(* IEC 61131-3 sources: beebread/doc (part 9) *)

// Commented out for beedance: it uses TN_INPUT_MENU_POPUP, which is commented out.
// FUNCTION_BLOCK TN_INPUT_SELECT_POPUP
// VAR
// 	in_index : INT;
// 	in_Element_Count : INT;
// 	by_Cur_Key : BYTE;
// 	by_Attr : BYTE;
// 	st_String : STRING;
// END_VAR
// VAR
// 	us_TN_MENU_POPUP : us_TN_MENU_POPUP;
// 	FB_TN_INPUT_MENU_POPUP : TN_INPUT_MENU_POPUP;
// 	FB_TN_SC_WRITE : TN_SC_WRITE;
// END_VAR
// VAR_IN_OUT
// 	Xus_TN_SCREEN : us_TN_SCREEN;
// 	Xus_TN_INPUT_CONTROL_DATA : us_TN_INPUT_CONTROL_DATA;
// END_VAR
//
// (* evaluate user input -> selection text n *)
// IF (Xus_TN_INPUT_CONTROL_DATA.bo_Focus = TRUE) THEN
//
// 	by_Cur_Key := Xus_TN_INPUT_CONTROL_DATA.by_Input_Exten_Code;
//
// 	IF (us_TN_MENU_POPUP.bo_Activ = FALSE) THEN
// 		us_TN_MENU_POPUP.by_Input_Exten_Code := BYTE#00;
//
// 		(* evaluate return key *)
// 		IF (by_Cur_Key = BYTE#13) THEN
// 			(* pass popup menu parameters *)
// 			us_TN_MENU_POPUP.in_Y := Xus_TN_INPUT_CONTROL_DATA.in_Y;
// 			us_TN_MENU_POPUP.in_X := Xus_TN_INPUT_CONTROL_DATA.in_X;
// 			us_TN_MENU_POPUP.by_Attr_mF := Xus_TN_INPUT_CONTROL_DATA.by_Attr_mF;
// 			us_TN_MENU_POPUP.by_Attr_oF := Xus_TN_INPUT_CONTROL_DATA.by_Attr_oF;
// 			us_TN_MENU_POPUP.st_Menu_Text := Xus_TN_INPUT_CONTROL_DATA.st_Input_Data;
// 			us_TN_MENU_POPUP.bo_Create := TRUE;
// 			us_TN_MENU_POPUP.in_Cur_Item := INT#00;
// 		END_IF;
//
// 		IF (us_TN_MENU_POPUP.in_Cur_Item > INT#00) THEN
// 			Xus_TN_INPUT_CONTROL_DATA.in_selected := us_TN_MENU_POPUP.in_Cur_Item;
// 			Xus_TN_INPUT_CONTROL_DATA.bo_Input_Entered := TRUE;
// 			Xus_TN_INPUT_CONTROL_DATA.bo_Update_Input := TRUE;
// 			us_TN_MENU_POPUP.in_Cur_Item := INT#00;
// 		END_IF;
//
// 	ELSE
// 		us_TN_MENU_POPUP.by_Input_Exten_Code := by_Cur_Key;
// 	END_IF;
//
// 	(* call popup menu cyclically *)
// 	FB_TN_INPUT_MENU_POPUP(Xus_TN_MENU_POPUP := us_TN_MENU_POPUP, Xus_TN_SCREEN := Xus_TN_SCREEN);
//
// END_IF;
//
// (* update of the display *)
// IF (Xus_TN_INPUT_CONTROL_DATA.bo_Update_Input = TRUE) OR (Xus_TN_INPUT_CONTROL_DATA.bo_Update_All = TRUE) THEN
//
// 	(* output title text *)
// 	IF Xus_TN_INPUT_CONTROL_DATA.bo_Update_All = TRUE THEN
//
// 		IF (Xus_TN_INPUT_CONTROL_DATA.in_Title_X_Offset = INT#00) AND (Xus_TN_INPUT_CONTROL_DATA.in_Title_Y_Offset = INT#00) THEN
// 			(* if offset X,Y = 0 then position the title string left of the element *)
// 			FB_TN_SC_WRITE.Iin_Y := Xus_TN_INPUT_CONTROL_DATA.in_Y;
// 			FB_TN_SC_WRITE.Iin_X := Xus_TN_INPUT_CONTROL_DATA.in_X - LEN(Xus_TN_INPUT_CONTROL_DATA.st_Title_String);
//
// 		ELSE
// 			(* output title text via row, color offset *)
// 			FB_TN_SC_WRITE.Iin_Y := Xus_TN_INPUT_CONTROL_DATA.in_Y + Xus_TN_INPUT_CONTROL_DATA.in_Title_Y_Offset;
// 			FB_TN_SC_WRITE.Iin_X := Xus_TN_INPUT_CONTROL_DATA.in_X + Xus_TN_INPUT_CONTROL_DATA.in_Title_X_Offset;
// 		END_IF;
//
// 		(* output title text via row, color offset *)
// 		FB_TN_SC_WRITE(	Iby_ATTR := Xus_TN_INPUT_CONTROL_DATA.by_Title_Attr,
// 						Ist_STRING := Xus_TN_INPUT_CONTROL_DATA.st_Title_String,
// 						Xus_TN_SCREEN := Xus_TN_SCREEN);
// 	END_IF;
//
// 	in_Element_Count := ELEMENT_COUNT(SEP:=BYTE#35,ELEMENT:=Xus_TN_INPUT_CONTROL_DATA.st_Input_Data);
//
// 	IF in_Element_Count > INT#00 THEN
//
// 		Xus_TN_INPUT_CONTROL_DATA.in_selected:=LIMIT(1,Xus_TN_INPUT_CONTROL_DATA.in_selected,in_Element_Count);
//
// 		in_index := Xus_TN_INPUT_CONTROL_DATA.in_selected;
//
// 		st_String := ELEMENT_GET(SEP:=BYTE#35,POS:=in_index - 1,ELEMENT:=Xus_TN_INPUT_CONTROL_DATA.st_Input_Data);
//
// 		st_String:= FIX(str:=st_String,
// 						L:=LEN(Xus_TN_INPUT_CONTROL_DATA.st_Input_Mask),
// 						C:=BYTE#32,
// 						M:=Xus_TN_INPUT_CONTROL_DATA.in_Input_Option);
//
// 		Xus_TN_INPUT_CONTROL_DATA.st_Input_String := st_String;
//
// 		IF Xus_TN_INPUT_CONTROL_DATA.bo_Focus = TRUE THEN
// 			by_Attr := Xus_TN_INPUT_CONTROL_DATA.by_Attr_mF;
// 		ELSE
// 			by_Attr := Xus_TN_INPUT_CONTROL_DATA.by_Attr_oF;
// 		END_IF;
//
// 		FB_TN_SC_WRITE(	Iin_X := Xus_TN_INPUT_CONTROL_DATA.in_X,
// 								Iin_Y := Xus_TN_INPUT_CONTROL_DATA.in_Y,
// 								Iby_ATTR := by_Attr,
// 								Ist_STRING := st_String,
// 								Xus_TN_SCREEN := Xus_TN_SCREEN );
// 	END_IF;
//
// 	(* set cursor to current position *)
// 	Xus_TN_INPUT_CONTROL_DATA.in_Cursor_X := Xus_TN_INPUT_CONTROL_DATA.in_X;
// 	Xus_TN_INPUT_CONTROL_DATA.in_Cursor_Y := Xus_TN_INPUT_CONTROL_DATA.in_Y;
//
// 	(* reset update flags *)
// 	Xus_TN_INPUT_CONTROL_DATA.bo_Update_All   := FALSE;
// 	Xus_TN_INPUT_CONTROL_DATA.bo_Update_Input := FALSE;
//
// END_IF;
// END_FUNCTION_BLOCK

// Commented out for beedance: it uses ELEMENT_COUNT, which is commented out.
// FUNCTION_BLOCK TN_INPUT_SELECT_TEXT
// VAR
// 	in_count : INT;
// 	by_Attr : BYTE;
// 	st_String : STRING;
// END_VAR
// VAR
// 	FB_TN_SC_WRITE : TN_SC_WRITE;
// END_VAR
// VAR_IN_OUT
// 	Xus_TN_SCREEN : us_TN_SCREEN;
// 	Xus_TN_INPUT_CONTROL_DATA : us_TN_INPUT_CONTROL_DATA;
// END_VAR
//
// (* evaluate user input -> selection text n *)
// IF Xus_TN_INPUT_CONTROL_DATA.bo_Focus = TRUE THEN
//
// (* evaluate space key *)
// 	IF Xus_TN_INPUT_CONTROL_DATA.by_Input_ASCII_Code = BYTE#32 THEN
// 		Xus_TN_INPUT_CONTROL_DATA.in_selected := Xus_TN_INPUT_CONTROL_DATA.in_selected + INT#01;
// 		Xus_TN_INPUT_CONTROL_DATA.bo_Update_Input := TRUE;
// 	END_IF;
//
// 	(* evaluate return key *)
// 	IF Xus_TN_INPUT_CONTROL_DATA.by_Input_Exten_Code = BYTE#13 THEN
// 		Xus_TN_INPUT_CONTROL_DATA.bo_Input_Entered := TRUE;
// 	END_IF;
//
// END_IF;
//
// (* update of the display *)
// IF (Xus_TN_INPUT_CONTROL_DATA.bo_Update_Input = TRUE) OR (Xus_TN_INPUT_CONTROL_DATA.bo_Update_All = TRUE) THEN
//
// 	(* output title text *)
// 	IF Xus_TN_INPUT_CONTROL_DATA.bo_Update_All = TRUE THEN
//
// 		IF (Xus_TN_INPUT_CONTROL_DATA.in_Title_X_Offset = INT#00) AND (Xus_TN_INPUT_CONTROL_DATA.in_Title_Y_Offset = INT#00) THEN
// 			(* if offset X,Y = 0 then position the title string left of the element *)
// 			FB_TN_SC_WRITE.Iin_Y := Xus_TN_INPUT_CONTROL_DATA.in_Y;
// 			FB_TN_SC_WRITE.Iin_X := Xus_TN_INPUT_CONTROL_DATA.in_X - LEN(Xus_TN_INPUT_CONTROL_DATA.st_Title_String);
//
// 		ELSE
// 			(* output title text via row, color offset *)
// 			FB_TN_SC_WRITE.Iin_Y := Xus_TN_INPUT_CONTROL_DATA.in_Y + Xus_TN_INPUT_CONTROL_DATA.in_Title_Y_Offset;
// 			FB_TN_SC_WRITE.Iin_X := Xus_TN_INPUT_CONTROL_DATA.in_X + Xus_TN_INPUT_CONTROL_DATA.in_Title_X_Offset;
// 		END_IF;
//
// 		(* output title text via row, color offset *)
// 		FB_TN_SC_WRITE(	Iby_ATTR := Xus_TN_INPUT_CONTROL_DATA.by_Title_Attr,
// 						Ist_STRING := Xus_TN_INPUT_CONTROL_DATA.st_Title_String,
// 						Xus_TN_SCREEN := Xus_TN_SCREEN);
//
// 	END_IF;
//
// 	(* process input line *)
//
// 	(* determine number of elements *)
// 	in_count := ELEMENT_COUNT(SEP:=BYTE#35,ELEMENT:=Xus_TN_INPUT_CONTROL_DATA.st_Input_Data);
//
// 	IF in_Count > INT#00 THEN
//
// 		IF Xus_TN_INPUT_CONTROL_DATA.in_selected < INT#1 THEN
// 			Xus_TN_INPUT_CONTROL_DATA.in_selected := INT#01;
// 		END_IF;
//
// 		IF Xus_TN_INPUT_CONTROL_DATA.in_selected > in_count THEN
// 			Xus_TN_INPUT_CONTROL_DATA.in_selected := INT#01;
// 		END_IF;
//
// 		st_String := ELEMENT_GET(SEP:=BYTE#35,POS:=Xus_TN_INPUT_CONTROL_DATA.in_selected - 1,ELEMENT:=Xus_TN_INPUT_CONTROL_DATA.st_Input_Data);
//
// 		st_String := FIX(	str:=st_String,
// 							L:=LEN(Xus_TN_INPUT_CONTROL_DATA.st_Input_Mask),
// 							C:=BYTE#32,
// 							M:=Xus_TN_INPUT_CONTROL_DATA.in_Input_Option);
//
// 		Xus_TN_INPUT_CONTROL_DATA.st_Input_String := st_String;
//
// 		IF Xus_TN_INPUT_CONTROL_DATA.bo_Focus = TRUE THEN
// 			by_Attr := Xus_TN_INPUT_CONTROL_DATA.by_Attr_mF;
// 		ELSE
// 			by_Attr := Xus_TN_INPUT_CONTROL_DATA.by_Attr_oF;
// 		END_IF;
//
// 		FB_TN_SC_WRITE(	Iin_Y := Xus_TN_INPUT_CONTROL_DATA.in_Y,
// 						Iin_X := Xus_TN_INPUT_CONTROL_DATA.in_X,
// 						Iby_ATTR := by_Attr,
// 						Ist_STRING := st_String,
// 						Xus_TN_SCREEN := Xus_TN_SCREEN);
// 	END_IF;
//
// 	(* set cursor to current position *)
// 	Xus_TN_INPUT_CONTROL_DATA.in_Cursor_Y := Xus_TN_INPUT_CONTROL_DATA.in_Y;
// 	Xus_TN_INPUT_CONTROL_DATA.in_Cursor_X := Xus_TN_INPUT_CONTROL_DATA.in_X;
//
// 	(* reset update flags *)
// 	Xus_TN_INPUT_CONTROL_DATA.bo_Update_All := FALSE;
// 	Xus_TN_INPUT_CONTROL_DATA.bo_Update_Input := FALSE;
//
// END_IF;
// END_FUNCTION_BLOCK

FUNCTION_BLOCK TN_RECEIVE
VAR_IN_OUT
	R_BUF :	NETWORK_BUFFER;
	Xus_TN_SCREEN : us_TN_SCREEN;
END_VAR
VAR
	REQ_Size : UINT;
	REQ1 : BYTE;
	REQ2 : BYTE;
	REQ3 : BYTE;
END_VAR

(* evaluate data reception *)
Xus_TN_SCREEN.by_Input_ASCII_Code := BYTE#00;
Xus_TN_SCREEN.by_Input_Exten_Code := BYTE#00;

IF R_BUF.SIZE > UINT#0 THEN
	(* evaluate received data *)
	REQ_Size := R_BUF.SIZE;
	REQ1 := R_BUF.BUFFER[0];
	REQ2 := R_BUF.BUFFER[1];
	REQ3 := R_BUF.BUFFER[2];

	IF REQ1 = BYTE#27 AND REQ_Size >= UINT#3 THEN (* Escape *)
		IF REQ2 = BYTE#91 THEN (* Cursor code *)
			IF (REQ3 >= BYTE#65 AND REQ3 <= BYTE#68) OR (REQ3 = BYTE#72) OR (REQ3 = BYTE#75) THEN (* 65..68 = cursor up,down,right,left / 72 = HOME / 75 = END *)
				Xus_TN_SCREEN.by_Input_Exten_Code := REQ3;
			END_IF;
		ELSIF REQ2 = BYTE#79 THEN (* special keys F1/F2/F3/F4 *)
			IF REQ3 >= BYTE#80 AND REQ3 <= BYTE#83 THEN
				Xus_TN_SCREEN.by_Input_Exten_Code := REQ3;
			END_IF;
		END_IF;
	ELSIF REQ1 >= BYTE#32 AND REQ1 <= BYTE#126 THEN
		Xus_TN_SCREEN.by_Input_ASCII_Code := REQ1;
		Xus_TN_SCREEN.bo_Input_ASCII_IsNum := ISC_NUM(REQ1); (* check for numeric input *)
	ELSIF REQ1 = BYTE#8 OR REQ1 = BYTE#9 OR REQ1 = BYTE#13 OR REQ1 = BYTE#27 THEN (* check for control characters 8=Backspace / 9=Tab / 13=Return / 27=Escape *)
		Xus_TN_SCREEN.by_Input_Exten_Code := REQ1;
	END_IF;

	(* set receive buffer data length to zero (destroy telegram *)
	R_BUF.SIZE := UINT#00;
END_IF;
END_FUNCTION_BLOCK

FUNCTION_BLOCK TN_SC_ADD_SHADOW
VAR
	in_Offset : INT;
	in_X : INT;
	in_Y : INT;
END_VAR
VAR_INPUT
	Iin_Y1 : INT;
	Iin_X1 : INT;
	Iin_Y2 : INT;
	Iin_X2 : INT;
	Iin_OPTION : INT;
END_VAR
VAR_IN_OUT
	Xus_TN_SCREEN : us_TN_SCREEN;
END_VAR

IF TN_SC_XY2_ERROR(Iin_X1,Iin_Y1,Iin_X2,Iin_Y2) THEN RETURN; END_IF;

IF Iin_Y1 < 0 OR Iin_X1 < 0 OR Iin_Y2 < 0 OR Iin_X2 < 0 THEN RETURN; END_IF; (* check min values *)
IF Iin_Y1 > 23 OR Iin_X1 > 79 OR Iin_Y2 > 23 OR Iin_X2 > 79 THEN RETURN; END_IF; (* check max values *)

in_Offset := (Iin_Y1 * 80) + Iin_X2;

IF Iin_OPTION = INT#00 THEN
	(* create shadow by adjusting color *)
	FOR in_Y := Iin_Y1 TO Iin_Y2 DO
		Xus_TN_SCREEN.bya_COLOR[in_Offset] := TN_SC_SHADOW_ATTR(Xus_TN_SCREEN.bya_COLOR[in_Offset]);
		in_Offset := in_Offset + 80;
		Xus_TN_SCREEN.bya_Line_Update[in_Y] := TRUE; (* mark line for update *)
	END_FOR;
ELSE
	(* create shadow with black color and spaces *)
	FOR in_Y := Iin_Y1 TO Iin_Y2 DO
		Xus_TN_SCREEN.bya_COLOR[in_Offset] := BYTE#00;
		Xus_TN_SCREEN.bya_CHAR[in_Offset] := BYTE#32;
		in_Offset := in_Offset + 80;
		Xus_TN_SCREEN.bya_Line_Update[in_Y] := TRUE; (* mark line for update *)
	END_FOR;
END_IF;

in_Offset := (Iin_Y2 * 80) + Iin_X1;

IF Iin_OPTION = INT#00 THEN
	(* create shadow by adjusting color *)
	FOR in_X  := Iin_X1 TO Iin_X2 DO
		Xus_TN_SCREEN.bya_COLOR[in_Offset] := TN_SC_SHADOW_ATTR(Xus_TN_SCREEN.bya_COLOR[in_Offset]);
		in_Offset := in_Offset + 1;
	END_FOR;
ELSE
	(* create shadow with black color and spaces *)
	FOR in_X  := Iin_X1 TO Iin_X2 DO
		Xus_TN_SCREEN.bya_COLOR[in_Offset] := BYTE#00;
		Xus_TN_SCREEN.bya_CHAR[in_Offset] := BYTE#32;
		in_Offset := in_Offset + 1;
	END_FOR;
END_IF;
END_FUNCTION_BLOCK

FUNCTION_BLOCK TN_SC_AREA_RESTORE
VAR
	in_Offset_1 : INT;
	in_Offset_2 : INT;
	in_Y : INT;
	in_X : INT;
	in_Y1 : INT;
	in_X1 : INT;
	in_Y2 : INT;
	in_X2 : INT;
END_VAR
VAR_IN_OUT
	Xus_TN_SCREEN : us_TN_SCREEN;
END_VAR

IF Xus_TN_SCREEN.bya_BACKUP[0] > BYTE#00 THEN

	(* read parameters *)
	in_X1 := BYTE_TO_INT(Xus_TN_SCREEN.bya_BACKUP[1]);
	in_Y1 := BYTE_TO_INT(Xus_TN_SCREEN.bya_BACKUP[2]);
	in_X2 := BYTE_TO_INT(Xus_TN_SCREEN.bya_BACKUP[3]);
	in_Y2 := BYTE_TO_INT(Xus_TN_SCREEN.bya_BACKUP[4]);

	IF TN_SC_XY2_ERROR(in_X1,in_Y1,in_X2,in_Y2) THEN RETURN; END_IF;
	in_Offset_2 := 5;

	(* restore CHAR and COLOR from BUFFER *)
	FOR in_Y := in_Y1 TO in_Y2 DO

		Xus_TN_SCREEN.bya_Line_Update[in_Y] := TRUE; (* release line for update *)
		in_Offset_1 := (in_Y * 80) + in_X1;

		FOR in_X := in_X1 TO in_X2 DO

			Xus_TN_SCREEN.bya_CHAR[in_Offset_1] := Xus_TN_SCREEN.bya_BACKUP[in_Offset_2];
			in_Offset_2 := in_Offset_2 + INT#01;

			Xus_TN_SCREEN.bya_COLOR[in_Offset_1] := Xus_TN_SCREEN.bya_BACKUP[in_Offset_2];
			in_Offset_2 := in_Offset_2 + INT#01;
			in_Offset_1 := in_Offset_1 + INT#01;

		END_FOR;
	END_FOR;

	(* mark data as invalid *)
	Xus_TN_SCREEN.bya_BACKUP[0] := BYTE#00;
END_IF;
END_FUNCTION_BLOCK

FUNCTION_BLOCK TN_SC_AREA_SAVE
VAR
	in_Offset_1 : INT;
	in_Offset_2 : INT;
	in_Y : INT;
	in_X : INT;
END_VAR
VAR_INPUT
	Iin_Y1 : INT;
	Iin_X1 : INT;
	Iin_Y2 : INT;
	Iin_X2 : INT;
END_VAR
VAR_IN_OUT
	Xus_TN_SCREEN : us_TN_SCREEN;
END_VAR

IF TN_SC_XY2_ERROR(Iin_X1,Iin_Y1,Iin_X2,Iin_Y2) THEN RETURN; END_IF;

(* store parameters *)
Xus_TN_SCREEN.bya_BACKUP[0] := BYTE#1;
Xus_TN_SCREEN.bya_BACKUP[1] := INT_TO_BYTE(Iin_X1);
Xus_TN_SCREEN.bya_BACKUP[2] := INT_TO_BYTE(Iin_Y1);
Xus_TN_SCREEN.bya_BACKUP[3] := INT_TO_BYTE(Iin_X2);
Xus_TN_SCREEN.bya_BACKUP[4] := INT_TO_BYTE(Iin_Y2);

in_Offset_2 := 5;
(* save CHAR and COLOR in BUFFER *)
FOR in_Y := Iin_Y1 TO Iin_Y2 DO

	in_Offset_1 := (in_Y * 80) + Iin_X1;
	FOR in_X := Iin_X1 TO Iin_X2 DO
		Xus_TN_SCREEN.bya_BACKUP[in_Offset_2] := Xus_TN_SCREEN.bya_CHAR[in_Offset_1];
		in_Offset_2 := in_Offset_2 + INT#01;
		Xus_TN_SCREEN.bya_BACKUP[in_Offset_2] := Xus_TN_SCREEN.bya_COLOR[in_Offset_1];
		in_Offset_2 := in_Offset_2 + INT#01;
		in_Offset_1 := in_Offset_1 + INT#01;
	END_FOR;
END_FOR;
END_FUNCTION_BLOCK

FUNCTION_BLOCK TN_SC_BOX
VAR
	FB_TN_SC_FILL : TN_SC_FILL;
	by_BorderChar_L_T : BYTE;
	by_BorderChar_T : BYTE;
	by_BorderChar_B : BYTE;
	by_BorderChar_R_T : BYTE;
	by_BorderChar_L : BYTE;
	by_BorderChar_R : BYTE;
	by_BorderChar_L_B : BYTE;
	by_BorderChar_R_B : BYTE;
	in_Y : INT;
	in_X : INT;
	in_Border_Offset : INT;
	in_Offset_1 : INT;
	in_Offset_2 : INT;
END_VAR
VAR_INPUT
	Iin_Y1 : INT;
	Iin_X1 : INT;
	Iin_Y2 : INT;
	Iin_X2 : INT;
	Iby_FILL : BYTE;
	Iby_ATTR : BYTE;
	Iin_BORDER : INT;
END_VAR
VAR_IN_OUT
	Xus_TN_SCREEN : us_TN_SCREEN;
END_VAR

IF TN_SC_XY2_ERROR(Iin_X1,Iin_Y1,Iin_X2,Iin_Y2) THEN RETURN; END_IF;

(* determine border type *)
CASE Iin_Border OF
0:
	in_Border_Offset := 0;
1:
	by_BorderChar_L_T := BYTE#218; (* top left *)
	by_BorderChar_T := BYTE#196; (* top *)
	by_BorderChar_R_T := BYTE#191; (* top right *)
	by_BorderChar_L := BYTE#179; (* left *)
	by_BorderChar_R := BYTE#179; (* right *)
	by_BorderChar_B := BYTE#196; (* bottom *)
	by_BorderChar_L_B := BYTE#217; (* bottom left *)
	by_BorderChar_R_B := BYTE#192; (* bottom right *)
	in_Border_Offset := 1;
 2:
	by_BorderChar_L_T := BYTE#201;
	by_BorderChar_T := BYTE#205;
	by_BorderChar_R_T := BYTE#187;
	by_BorderChar_L := BYTE#186;
	by_BorderChar_R := BYTE#186;
	by_BorderChar_B := BYTE#205;
	by_BorderChar_L_B := BYTE#188;
	by_BorderChar_R_B := BYTE#200;
	in_Border_Offset := 1;
ELSE
	by_BorderChar_L_T := BYTE#32;
	by_BorderChar_T := BYTE#32;
	by_BorderChar_R_T := BYTE#32;
	by_BorderChar_L := BYTE#32;
	by_BorderChar_R := BYTE#32;
	by_BorderChar_B := BYTE#32;
	by_BorderChar_L_B := BYTE#32;
	by_BorderChar_R_B := BYTE#32;
	in_Border_Offset := 1;

END_CASE;

IF Iby_FILL > BYTE#0 THEN (* FILL character present? -> draw box *)

	(* draw fill function one character row smaller *)
	FB_TN_SC_FILL(	Iin_Y1 := Iin_Y1 + in_Border_Offset,
					Iin_X1 := Iin_X1 + in_Border_Offset,
					Iin_Y2 := Iin_Y2 - in_Border_Offset,
					Iin_X2 := Iin_X2 - in_Border_Offset,
					Iby_CHAR := Iby_FILL,
					Iby_Attr := Iby_ATTR,
					Xus_TN_SCREEN := Xus_TN_SCREEN);
END_IF;

IF Iin_BORDER = 0 THEN RETURN; END_IF;

(* output left and right border *)

in_Offset_1 := (Iin_Y1 * 80) + Iin_X1;
in_Offset_2 := (Iin_Y1 * 80) + Iin_X2;

FOR in_Y := Iin_Y1 TO Iin_Y2 DO

	(* release line for update *)
	Xus_TN_SCREEN.bya_Line_Update[in_Y] := TRUE;

	Xus_TN_SCREEN.bya_CHAR[in_Offset_1] := by_BorderChar_L;
	Xus_TN_SCREEN.bya_COLOR[in_Offset_1] := Iby_Attr;

	Xus_TN_SCREEN.bya_CHAR[in_Offset_2] := by_BorderChar_R;
	Xus_TN_SCREEN.bya_COLOR[in_Offset_2] := Iby_Attr;

	in_Offset_1 := in_Offset_1 + 80;
	in_Offset_2 := in_Offset_2 + 80;

END_FOR;

(* output bottom and top border *)
in_Offset_1 := (Iin_Y1 * 80) + Iin_X1;
in_Offset_2 := (Iin_Y2 * 80) + Iin_X1;

FOR in_X := Iin_X1 TO Iin_X2 DO

	Xus_TN_SCREEN.bya_CHAR[in_Offset_1] := by_BorderChar_T;
	Xus_TN_SCREEN.bya_COLOR[in_Offset_1] := Iby_Attr;

	Xus_TN_SCREEN.bya_CHAR[in_Offset_2] := by_BorderChar_B;
	Xus_TN_SCREEN.bya_COLOR[in_Offset_2] := Iby_Attr;

	in_Offset_1 := in_Offset_1 + INT#1;
	in_Offset_2 := in_Offset_2 + INT#1;

END_FOR;

(* output top left corner *)
in_Offset_1 := (Iin_Y1 * 80) + Iin_X1;
Xus_TN_SCREEN.bya_CHAR[in_Offset_1] := by_BorderChar_L_T;
Xus_TN_SCREEN.bya_COLOR[in_Offset_1] := Iby_Attr;

(* output top right corner *)
in_Offset_1 := (Iin_Y1 * 80) + Iin_X2;
Xus_TN_SCREEN.bya_CHAR[in_Offset_1] := by_BorderChar_R_T;
Xus_TN_SCREEN.bya_COLOR[in_Offset_1] := Iby_Attr;

(* output bottom left corner *)
in_Offset_1 := (Iin_Y2 * 80) + Iin_X1;
Xus_TN_SCREEN.bya_CHAR[in_Offset_1] := by_BorderChar_R_B;
Xus_TN_SCREEN.bya_COLOR[in_Offset_1] := Iby_Attr;

(* output bottom right corner *)
in_Offset_1 := (Iin_Y2 * 80) + Iin_X2;
Xus_TN_SCREEN.bya_CHAR[in_Offset_1] := by_BorderChar_L_B;
Xus_TN_SCREEN.bya_COLOR[in_Offset_1] := Iby_Attr;
END_FUNCTION_BLOCK

FUNCTION_BLOCK TN_SC_FILL
VAR
	in_X : INT;
	in_Y : INT;
	in_Offset : INT;
END_VAR
VAR_INPUT
	Iin_Y1 : INT;
	Iin_X1 : INT;
	Iin_Y2 : INT;
	Iin_X2 : INT;
	Iby_CHAR : BYTE;
	Iby_Attr : BYTE;
END_VAR
VAR_IN_OUT
	Xus_TN_SCREEN : us_TN_SCREEN;
END_VAR

IF TN_SC_XY2_ERROR(Iin_X1,Iin_Y1,Iin_X2,Iin_Y2) THEN RETURN; END_IF;

FOR in_Y := Iin_Y1 TO Iin_Y2 DO
	Xus_TN_SCREEN.bya_Line_Update[in_Y] := TRUE; (* release line for update *)
	in_Offset := (in_Y * 80) + Iin_X1;
	FOR in_X := Iin_X1 TO Iin_X2 DO
		Xus_TN_SCREEN.bya_CHAR[in_Offset]  := Iby_CHAR; (* enter character *)
		Xus_TN_SCREEN.bya_COLOR[in_Offset] := Iby_Attr; (* enter color *)
		in_Offset := in_Offset + 1;
	END_FOR;
END_FOR;
END_FUNCTION_BLOCK

FUNCTION_BLOCK TN_SC_LINE
VAR
	by_Connect_Left_Char : BYTE;
	by_Connect_Right_Char : BYTE;
	by_Connect_Top_Char : BYTE;
	by_Connect_Bottom_Char : BYTE;
	by_Connect_Cruz_Char : BYTE;
	by_Vertikal_Line_Char : BYTE;
	by_Horzontal_Line_Char : BYTE;
	by_old_Char : BYTE;
	in_Offset_1 : INT;
	in_ROW_Index : INT;
	in_COL_Index : INT;
	by_Char : BYTE;
END_VAR
VAR_INPUT
	Iin_X1 : INT;
	Iin_Y1 : INT;
	Iin_X2 : INT;
	Iin_Y2 : INT;
	Iby_ATTR : BYTE;
	Iby_BORDER : BYTE;
END_VAR
VAR_IN_OUT
	Xus_TN_SCREEN : us_TN_SCREEN;
END_VAR

IF TN_SC_XY2_ERROR(Iin_X1,Iin_Y1,Iin_X2,Iin_Y2) THEN RETURN; END_IF;

(* determine border type *)
IF Iby_Border = BYTE#01 THEN (* Single Line *)
	by_Connect_Top_Char := BYTE#16#C2;
	by_Connect_Bottom_Char := BYTE#16#C1;
	by_Connect_Left_Char := BYTE#16#C3;
	by_Connect_Right_Char := BYTE#16#B4;
	by_Horzontal_Line_Char := BYTE#16#C4;
	by_Vertikal_Line_Char := BYTE#16#B3;
	by_Connect_Cruz_Char := BYTE#16#C5;
ELSIF Iby_Border = BYTE#02 THEN	(* double line *)
	by_Connect_Top_Char := BYTE#16#CB;
	by_Connect_Bottom_Char := BYTE#16#CA;
	by_Connect_Left_Char := BYTE#16#CC;
	by_Connect_Right_Char := BYTE#16#B9;
	by_Horzontal_Line_Char := BYTE#16#CD;
	by_Vertikal_Line_Char := BYTE#16#BA;
	by_Connect_Cruz_Char := BYTE#16#CE;
ELSE (* full line *)
	by_Connect_Top_Char := Iby_Border;
	by_Connect_Bottom_Char := Iby_Border;
	by_Connect_Left_Char := Iby_Border;
	by_Connect_Right_Char := Iby_Border;
	by_Horzontal_Line_Char := Iby_Border;
	by_Vertikal_Line_Char := Iby_Border;
	by_Connect_Cruz_Char := Iby_Border;
END_IF;

(* draw vertical line *)
IF Iin_X1 = Iin_X2 THEN
	in_Offset_1 := (Iin_Y1 * 80) + Iin_X1;
	FOR in_ROW_Index := Iin_Y1 TO Iin_Y2 DO
		by_old_Char := Xus_TN_SCREEN.bya_CHAR[in_Offset_1]; (* read existing character *)
		by_Char := by_Vertikal_Line_Char; (* preset default characters *)
		IF by_old_Char = by_Horzontal_Line_Char THEN (* intersection detected *)
			IF in_ROW_Index = Iin_Y1 THEN (* handle start of line *)
				by_Char := by_Connect_Top_Char;
			ELSIF in_ROW_Index = Iin_Y2 THEN (* handle end of line *)
				by_Char := by_Connect_Bottom_Char;
			ELSE (* handle crossing point *)
				by_Char := by_Connect_Cruz_Char;
			END_IF;
		END_IF;
		Xus_TN_SCREEN.bya_Line_Update[in_ROW_Index] := TRUE; (* release line for update *)
		Xus_TN_SCREEN.bya_CHAR[in_Offset_1] := by_Char;
		Xus_TN_SCREEN.bya_COLOR[in_Offset_1] := Iby_Attr;
		in_Offset_1 := in_Offset_1 + 80;
	END_FOR;

ELSIF Iin_Y1 = Iin_Y2 THEN (* draw horizontal line *)
	Xus_TN_SCREEN.bya_Line_Update[Iin_Y1] := TRUE; (* release line for update *)
	in_Offset_1 := (Iin_Y1 * 80) + Iin_X1;
	FOR in_COL_Index := Iin_X1 TO Iin_X2 DO
		by_old_Char := Xus_TN_SCREEN.bya_CHAR[in_Offset_1]; (* read existing character *)
		by_Char := by_Horzontal_Line_Char; (* preset default characters *)
		IF by_old_Char = by_Vertikal_Line_Char THEN (* intersection detected *)
			IF in_COL_Index = Iin_X1 THEN (* handle start of line *)
				by_Char := by_Connect_Left_Char;
			ELSIF in_COL_Index = Iin_X2 THEN (* handle end of line *)
				by_Char := by_Connect_Right_Char;
			ELSE (* handle crossing point *)
				by_Char := by_Connect_Cruz_Char;
			END_IF;
		END_IF;
		Xus_TN_SCREEN.bya_CHAR[in_Offset_1] := by_Char;
		Xus_TN_SCREEN.bya_COLOR[in_Offset_1] := Iby_Attr;
		in_Offset_1 := in_Offset_1 + 1;
	END_FOR;
END_IF;
END_FUNCTION_BLOCK

FUNCTION_BLOCK TN_SC_READ_ATTR
VAR
	in_Offset : INT;
END_VAR
VAR_INPUT
	Iin_Y : INT;
	Iin_X : INT;
END_VAR
VAR_OUTPUT
	Oby_ATTR : BYTE;
END_VAR
VAR_IN_OUT
	Xus_TN_SCREEN : us_TN_SCREEN;
END_VAR

IF TN_SC_XY_ERROR(Iin_X,Iin_Y) THEN RETURN; END_IF;
in_Offset := (Iin_Y * 80) + Iin_X;
Oby_ATTR := Xus_TN_SCREEN.bya_COLOR[in_Offset]; (* read attributes *)
END_FUNCTION_BLOCK

FUNCTION_BLOCK TN_SC_READ_CHAR
VAR
	in_Offset : INT;
END_VAR
VAR_INPUT
	Iin_Y : INT;
	Iin_X : INT;
END_VAR
VAR_OUTPUT
	Oby_CHAR : BYTE;
END_VAR
VAR_IN_OUT
	Xus_TN_SCREEN : us_TN_SCREEN;
END_VAR

IF TN_SC_XY_ERROR(Iin_X,Iin_Y) THEN RETURN; END_IF;
in_Offset := (Iin_Y * 80) + Iin_X;
Oby_CHAR := Xus_TN_SCREEN.bya_CHAR[in_Offset]; (* read character *)
END_FUNCTION_BLOCK

FUNCTION TN_SC_SHADOW_ATTR : BYTE
VAR_INPUT
	Iby_ATTR : BYTE;
END_VAR

(* change background color to black      *)
(* and switch on dark foreground colors *)
TN_SC_SHADOW_ATTR := ((Iby_ATTR AND BYTE#2#11110000) OR BYTE#2#00001000);
END_FUNCTION

// Commented out for beedance: it uses FIX, which is commented out.
// FUNCTION_BLOCK TN_SC_VIEWPORT
// VAR
// 	FB_TN_SC_WRITE : TN_SC_WRITE;
// 	FB_TON : TON;
// END_VAR
// VAR
// 	in_index : INT;
// 	in_Color : INT;
// 	by_Attr : BYTE;
// 	in_count : INT;
// END_VAR
// VAR_IN_OUT
// 	Xus_LOG_VIEWPORT : us_LOG_VIEWPORT;
// 	Xus_LOG_CONTROL : LOG_CONTROL;
// 	Xus_TN_SCREEN : us_TN_SCREEN;
// END_VAR
// VAR_INPUT
// 	Iin_X : INT;
// 	Iin_Y : INT;
// 	Iin_Width : INT;
// 	Idw_ATTR_1 : DWORD;
// 	Idw_ATTR_2 : DWORD;
// 	Iti_TIME : TIME;
// END_VAR
//
// (* output LOG messages *)
//
// IF Xus_LOG_VIEWPORT.UPDATE AND FB_TON.Q THEN (* update requested and delay time elapsed *)
// 	Xus_LOG_VIEWPORT.UPDATE := FALSE;
// 	FOR in_count := 1 TO Xus_LOG_VIEWPORT.COUNT DO (* process all viewport lines *)
// 		in_index := Xus_LOG_VIEWPORT.LINE_ARRAY[in_count];
// 		(* read color from the option parameter >0,Level,Back,Front< *)
// 		in_Color := DWORD_TO_INT(Xus_LOG_CONTROL.MSG_OPTION[in_index] AND DWORD#2#1111);
//
// 		CASE in_Color OF
// 		0..3: by_Attr := BYTE_OF_DWORD(Idw_ATTR_1,INT_TO_BYTE(in_Color));
// 		4..7: by_Attr := BYTE_OF_DWORD(Idw_ATTR_2,INT_TO_BYTE(in_Color));
// 		ELSE
// 			by_Attr := BYTE_OF_DWORD(Idw_ATTR_1,BYTE#0);
// 		END_CASE;
//
// 		(* output message (text + color) *)
// 		FB_TN_SC_WRITE(	Iin_Y := Iin_Y + in_count - INT#01,
// 						Iin_X := Iin_X,
// 						Iby_ATTR := by_Attr,
// 						Ist_STRING := FIX(str := Xus_LOG_CONTROL.MSG[in_index], L := Iin_Width, C := BYTE#32, M := INT#00), (* pad or truncate string on the right *)
// 						Xus_TN_SCREEN := Xus_TN_SCREEN);
//
// 	END_FOR;
//
// 	(* stop/reset timer *)
// 	FB_TON.IN := FALSE;
// 	FB_TON.PT := Iti_TIME;
// 	FB_TON();
//
// END_IF;
//
// (* update time delay *)
// FB_TON.IN := TRUE;
// FB_TON.PT := Iti_TIME;
// FB_TON();
// END_FUNCTION_BLOCK

// Commented out for beedance: it uses CODE, which is commented out.
// FUNCTION_BLOCK TN_SC_WRITE
// VAR
// 	bo_Color : BOOL;
// 	in_Offset : INT;
// 	in_Char_Index : INT;
// 	in_String_Length : INT;
// END_VAR
// VAR_INPUT
// 	Iin_Y : INT;
// 	Iin_X : INT;
// 	Iby_ATTR : BYTE;
// 	Ist_STRING : STRING;
// END_VAR
// VAR_IN_OUT
// 	Xus_TN_SCREEN : us_TN_SCREEN;
// END_VAR
//
// in_String_Length := LEN(Ist_STRING);
// IF TN_SC_XY_ERROR(Iin_X + in_String_Length - 1,Iin_Y) THEN RETURN; END_IF;
// Xus_TN_SCREEN.bya_Line_Update[Iin_Y] := TRUE; (* release line for update *)
// in_Offset := (Iin_Y * 80) + Iin_X; (* calculate offset of the first character *)
// bo_Color := Iby_ATTR <> BYTE#00;
//
// (* copy characters and attributes of the string *)
// FOR in_Char_Index := 1 TO in_String_Length DO
// 	IF bo_Color THEN Xus_TN_SCREEN.bya_COLOR[in_Offset] := Iby_ATTR; END_IF;
// 	Xus_TN_SCREEN.bya_CHAR[in_Offset] := CODE(STR:=Ist_STRING,POS:=in_Char_Index);
// 	in_Offset := in_Offset + INT#1;
// END_FOR;
//
// Xus_TN_SCREEN.in_EOS_Offset := in_Offset; (* save end of string offset *)
// END_FUNCTION_BLOCK

FUNCTION_BLOCK TN_SC_WRITE_ATTR
VAR
	in_Offset : INT;
END_VAR
VAR_INPUT
	Iin_Y : INT;
	Iin_X : INT;
	Iby_ATTR : BYTE;
END_VAR
VAR_IN_OUT
	Xus_TN_SCREEN : us_TN_SCREEN;
END_VAR

IF TN_SC_XY_ERROR(Iin_X,Iin_Y) THEN RETURN; END_IF;
in_Offset := (Iin_Y * 80) + Iin_X;
Xus_TN_SCREEN.bya_COLOR[in_Offset] := Iby_ATTR; (* write attributes *)
END_FUNCTION_BLOCK

// Commented out for beedance: it uses TN_SC_WRITE, which is commented out.
// FUNCTION_BLOCK TN_SC_WRITE_C
// VAR
// 	FB_TN_SC_WRITE : TN_SC_WRITE;
// END_VAR
// VAR_INPUT
// 	Iin_Y : INT;
// 	Iin_X : INT;
// 	Iby_ATTR : BYTE;
// 	Ist_STRING : STRING;
// 	Iin_LENGTH : INT;
// 	Iin_OPTION : INT;
// END_VAR
// VAR_IN_OUT
// 	Xus_TN_SCREEN : us_TN_SCREEN;
// END_VAR
//
// (* output text *)
// FB_TN_SC_WRITE( Iin_Y := Iin_Y,
// 				Iin_X := Iin_X,
// 				Iby_ATTR := Iby_ATTR,
// 				Ist_STRING := FIX(str:=Ist_STRING,L:=Iin_LENGTH,C:=BYTE#32,M:=Iin_OPTION),
// 				Xus_TN_SCREEN := Xus_TN_SCREEN);
// END_FUNCTION_BLOCK

FUNCTION_BLOCK TN_SC_WRITE_CHAR
VAR
	in_Offset : INT;
END_VAR
VAR_INPUT
	Iin_Y : INT;
	Iin_X : INT;
	Iby_CHAR : BYTE;
END_VAR
VAR_IN_OUT
	Xus_TN_SCREEN : us_TN_SCREEN;
END_VAR

IF TN_SC_XY_ERROR(Iin_X,Iin_Y) THEN RETURN; END_IF;
in_Offset := (Iin_Y * 80) + Iin_X;
Xus_TN_SCREEN.bya_CHAR[in_Offset] := Iby_CHAR; (* write character *)
END_FUNCTION_BLOCK

FUNCTION_BLOCK TN_SC_WRITE_EOS
VAR
	TN_SC_WRITE : TN_SC_WRITE;
END_VAR
VAR_INPUT
	Iby_ATTR : BYTE;
	Ist_STRING : STRING;
END_VAR
VAR_IN_OUT
	Xus_TN_SCREEN : us_TN_SCREEN;
END_VAR

TN_SC_WRITE(Iin_Y := Xus_TN_SCREEN.in_EOS_Offset / 80, (* calculate current line *)
			Iin_X := Xus_TN_SCREEN.in_EOS_Offset MOD 80, (* calculate current column *)
			Iby_ATTR := Iby_ATTR,
			Ist_STRING := Ist_STRING,
			Xus_TN_SCREEN := Xus_TN_SCREEN);
END_FUNCTION_BLOCK

FUNCTION TN_SC_XY2_ERROR : BOOL
VAR_INPUT
	X1 : INT;
	Y1 : INT;
	X2 : INT;
	Y2 : INT;
END_VAR

(* check min and max values *)
TN_SC_XY2_ERROR := Y1 < 0 OR X1 < 0 OR Y2 < 0 OR X2 < 0 OR Y1 > 23 OR X1 > 79 OR Y2 > 23 OR X2 > 79;
END_FUNCTION

FUNCTION TN_SC_XY_ERROR : BOOL
VAR_INPUT
	X : INT;
	Y : INT;
END_VAR

(* check min and max values *)
TN_SC_XY_ERROR := Y < 0 OR X < 0 OR Y > 23 OR X > 79;
END_FUNCTION

FUNCTION_BLOCK TN_SEND_ROWS
VAR_IN_OUT
	IP_C : IP_C;
	S_BUF : NETWORK_BUFFER;
	Xus_TN_SCREEN : us_TN_SCREEN;
END_VAR
VAR_INPUT
	S_BUF_SIZE : INT;
END_VAR
VAR
	in_Line_Count : INT;(*counter to run through at most all 24 lines*)
	in_Col_Count : INT;
	in_Last_Row_Index : INT;
	bo_Break_Loop : BOOL;
	in_Row_Count : INT;
	in_Offset : INT;
	in_Write_Index : INT;
	in_Write_Index_Backup : INT;
	by_Cur_Color : BYTE;
	by_last_Color : BYTE;
	in_Write_Stop : INT;
END_VAR

(* connection present and no data sending active *)
IF (IP_C.C_STATE < BYTE#127 OR S_BUF.SIZE > UINT#0) THEN
	RETURN; (* no -> exit block *)
END_IF;

(* load current write index *)
in_Write_Index := UINT_TO_INT(S_BUF.SIZE) - 1;

(* buffer current write index *)
in_Write_Index_Backup := in_Write_Index;

(* rising edge connect on *)
IF (IP_C.C_STATE = BYTE#254) OR (Xus_TN_SCREEN.bo_Clear_Screen) THEN

	(* reset clear-screen message *)
	Xus_TN_SCREEN.bo_Clear_Screen := FALSE;

	(* mark all lines for update *)
	FOR in_Line_Count := INT#00 TO INT#23 DO
		Xus_TN_SCREEN.bya_Line_Update[in_Line_Count] := TRUE;
	END_FOR;

	(* ESC [0;30,40m  Reset Attributes + Black,Black *)
	in_Write_Index := in_Write_Index + INT#1;
	S_BUF.BUFFER[in_Write_Index] := BYTE#16#1B; (* ESC *)
	in_Write_Index := in_Write_Index + INT#1;
	S_BUF.BUFFER[in_Write_Index] := BYTE#16#5B; (* [ *)
	in_Write_Index := in_Write_Index + INT#1;
	S_BUF.BUFFER[in_Write_Index] := BYTE#16#30; (* 0 *)
	in_Write_Index := in_Write_Index + INT#1;
	S_BUF.BUFFER[in_Write_Index] := BYTE#16#3B; (* ; *)
	in_Write_Index := in_Write_Index + INT#1;
	S_BUF.BUFFER[in_Write_Index] := BYTE#16#33; (* 3 *)

	(* output ones digit of foreground color *)
	in_Write_Index := in_Write_Index + INT#1;
	S_BUF.BUFFER[in_Write_Index] := (SHR(Xus_TN_SCREEN.by_Clear_Screen_Attr,4) OR BYTE#16#30);

	in_Write_Index := in_Write_Index + INT#1;
	S_BUF.BUFFER[in_Write_Index] := BYTE#16#3B; (* ; *)
	in_Write_Index := in_Write_Index + INT#1;
	S_BUF.BUFFER[in_Write_Index] := BYTE#16#34; (* 4 *)

	(* output ones digit of background color *)
	in_Write_Index := in_Write_Index + INT#1;
	S_BUF.BUFFER[in_Write_Index] := ((Xus_TN_SCREEN.by_Clear_Screen_Attr AND BYTE#16#07) OR BYTE#16#30);

	in_Write_Index := in_Write_Index + INT#1;
	S_BUF.BUFFER[in_Write_Index] := BYTE#16#6D; (* m *)

	(* ESC[2J Clear screen and home cursor *)
	in_Write_Index := in_Write_Index + INT#1;
	S_BUF.BUFFER[in_Write_Index] := BYTE#16#1B; (* ESC *)
	in_Write_Index := in_Write_Index + INT#1;
	S_BUF.BUFFER[in_Write_Index] := BYTE#16#5B; (* [ *)
	in_Write_Index := in_Write_Index + INT#1;
	S_BUF.BUFFER[in_Write_Index] := BYTE#16#32; (* 2 *)
	in_Write_Index := in_Write_Index + INT#1;
	S_BUF.BUFFER[in_Write_Index] := BYTE#16#4A; (* J *)

	(* ESC [?7l Off *)
	in_Write_Index := in_Write_Index + INT#1;
	S_BUF.BUFFER[in_Write_Index] := BYTE#16#1B; (* ESC *)
	in_Write_Index := in_Write_Index + INT#1;
	S_BUF.BUFFER[in_Write_Index] := BYTE#16#5B; (* [ *)
	in_Write_Index := in_Write_Index + INT#1;
	S_BUF.BUFFER[in_Write_Index] := BYTE#16#3F; (* ? *)
	in_Write_Index := in_Write_Index + INT#1;
	S_BUF.BUFFER[in_Write_Index] := BYTE#16#37; (* 7 *)
	in_Write_Index := in_Write_Index + INT#1;
	S_BUF.BUFFER[in_Write_Index] := BYTE#16#6C; (* l *)

END_IF;

in_Last_Row_Index := INT#0;
bo_Break_Loop := FALSE;
in_Write_Stop := S_BUF_SIZE - 20;

(* run through all lines *)
FOR in_Line_Count := 0 TO 23 DO

	in_Offset := in_Row_Count * INT#80;

	(* check whether an update of a line is necessary, or after reconnect *)
	IF (Xus_TN_SCREEN.bya_Line_Update[in_Row_Count] = TRUE) THEN

		(* position write cursor *)
		in_Write_Index := in_Write_Index + INT#1;
		S_BUF.BUFFER[in_Write_Index] := BYTE#16#1B; (* ESC *)
		in_Write_Index := in_Write_Index + INT#1;
		S_BUF.BUFFER[in_Write_Index] := BYTE#16#5B; (* [ *)

		(* output tens digit of line number *)
		in_Write_Index := in_Write_Index + INT#1;
		S_BUF.BUFFER[in_Write_Index] :=
		SHR(INT_TO_BCDC(in_Row_Count + INT#1),INT#4) OR BYTE#16#30;

		(* output ones digit of line number *)
		in_Write_Index := in_Write_Index + INT#1;
		S_BUF.BUFFER[in_Write_Index] :=
		(INT_TO_BCDC(in_Row_Count + INT#1) AND BYTE#16#0F) OR BYTE#16#30;

		in_Write_Index := in_Write_Index + INT#1;
		S_BUF.BUFFER[in_Write_Index] := BYTE#16#3B; (* ; *)
		in_Write_Index := in_Write_Index + INT#1;
		S_BUF.BUFFER[in_Write_Index] := BYTE#16#31; (* 1 *)
		in_Write_Index := in_Write_Index + INT#1;
		S_BUF.BUFFER[in_Write_Index] := BYTE#16#48; (* H *)

		(* run through all columns of a line *)
		FOR in_Col_Count := 0 TO 79 DO

			(* determine current color *)
			by_Cur_Color := Xus_TN_SCREEN.bya_COLOR[in_Offset];
			IF (by_Cur_Color <> by_last_Color) OR (in_Col_Count = INT#00) THEN

				(* color setting: output ANSI sequence ESC[X;Y;Zm *)
				in_Write_Index := in_Write_Index + INT#1;
				S_BUF.BUFFER[in_Write_Index] := BYTE#16#1B; (* ESC *)

				in_Write_Index := in_Write_Index + INT#1;
				S_BUF.BUFFER[in_Write_Index] := BYTE#16#5B; (* [ *)

				(* color setting: determine dark or bright and blinking *)

					IF (((by_Cur_Color AND BYTE#2#10001000) XOR (by_last_Color AND BYTE#2#10001000)) <> BYTE#00) OR (in_Col_Count = 0) THEN

						in_Write_Index := in_Write_Index + INT#1;
						S_BUF.BUFFER[in_Write_Index] := BYTE#16#30; (* 0 *)
						in_Write_Index := in_Write_Index + INT#1;
						S_BUF.BUFFER[in_Write_Index] := BYTE#16#3B; (* ; *)

						(* no dark colors wanted -> then bold & bright *)
						IF (by_Cur_Color AND BYTE#2#00001000) = BYTE#2#00000000 THEN

							(* switch to bold & bright colors *)
							in_Write_Index := in_Write_Index + INT#1;
							S_BUF.BUFFER[in_Write_Index] := BYTE#16#31; (* 1 *)
							in_Write_Index := in_Write_Index + INT#1;
							S_BUF.BUFFER[in_Write_Index] := BYTE#16#3B; (* ; *)

						END_IF;

						(* blinking colors wanted *)
						IF (by_Cur_Color AND BYTE#2#10000000) = BYTE#2#10000000 THEN

							(* switch to bold & bright colors *)
							in_Write_Index := in_Write_Index + INT#1;
							S_BUF.BUFFER[in_Write_Index] := BYTE#16#35; (* 5 *)
							in_Write_Index := in_Write_Index + INT#1;
							S_BUF.BUFFER[in_Write_Index] := BYTE#16#3B; (* ; *)

						END_IF;

					END_IF;

					(* output tens digit of foreground color *)
					in_Write_Index := in_Write_Index + INT#1;
					S_BUF.BUFFER[in_Write_Index] := BYTE#16#33; (* 3 *)

					(* output ones digit of foreground color *)
					in_Write_Index := in_Write_Index + INT#1;
					S_BUF.BUFFER[in_Write_Index] := ((SHR(by_Cur_Color,4) AND BYTE#2#00000111) OR BYTE#16#30);

					in_Write_Index := in_Write_Index + INT#1;
					S_BUF.BUFFER[in_Write_Index] := BYTE#16#3B; (* ; *)

					(* output tens digit of background color *)
					in_Write_Index := in_Write_Index + INT#1;
					S_BUF.BUFFER[in_Write_Index] := BYTE#16#34; (* 4 *)

					(* output ones digit of background color *)
					in_Write_Index := in_Write_Index + INT#1;
					S_BUF.BUFFER[in_Write_Index] := ((by_Cur_Color AND BYTE#2#00000111) OR BYTE#16#30);

					in_Write_Index := in_Write_Index + INT#1;
					S_BUF.BUFFER[in_Write_Index] := BYTE#16#6D; (* m *)

					(* store new color as last used *)
					by_last_Color := by_Cur_Color;

				END_IF;

				(* end of buffer reached early -> end *)
				IF (in_Write_Index > in_Write_Stop) THEN

					bo_Break_Loop := TRUE;
					EXIT;

				END_IF;

				(* transfer one TEXT character from the screen buffer to the send buffer *)
				in_Write_Index := in_Write_Index + INT#1;
				S_BUF.BUFFER[in_Write_Index] := Xus_TN_SCREEN.bya_CHAR[in_Offset];

				(* select next column *)
				in_Offset := in_Offset + INT#01;
			END_FOR;

			IF (bo_Break_Loop = TRUE) THEN;

				(* end of buffer reached early -> transfer only up to the last complete line *)
				in_Write_Index := in_Last_Row_Index;

				EXIT;
			END_IF;

			(* buffer is not full yet -> take new line *)
			in_Last_Row_Index := in_Write_Index;
			Xus_TN_SCREEN.bya_Line_Update[in_Row_Count] := FALSE;

		END_IF;

		(* address next line *)
		in_Row_Count := in_Row_Count + INT#01;

		(* after the last line start again from the beginning *)
		IF (in_Row_Count > INT#23) THEN
			in_Row_Count := INT#00;
		END_IF;
		(*-----------------------------------------------*)

	END_FOR;

	(* if all lines were done at once in one update cycle *)
	(* Row_Count is set to the first line *)
	(* meant to prevent ugly graphics flicker *)
	(* otherwise continue at the last line *)
	IF (bo_Break_Loop = FALSE) THEN
		in_Row_Count := INT#00;
	END_IF;

	(* position edit cursor *)
	IF (in_Write_Index <> in_Write_Index_Backup) THEN

		in_Write_Index := in_Write_Index + INT#1;
		S_BUF.BUFFER[in_Write_Index] := BYTE#16#1B; (* ESC *)
		in_Write_Index := in_Write_Index + INT#1;
		S_BUF.BUFFER[in_Write_Index] := BYTE#16#5B; (* [ *)

		(* output tens digit of line number *)
		in_Write_Index := in_Write_Index + INT#1;
		S_BUF.BUFFER[in_Write_Index] := SHR(INT_TO_BCDC(Xus_TN_SCREEN.in_Cursor_Y + 1),INT#4) OR BYTE#16#30;

		(* output ones digit of line number *)
		in_Write_Index := in_Write_Index + INT#1;
		S_BUF.BUFFER[in_Write_Index] := (INT_TO_BCDC(Xus_TN_SCREEN.in_Cursor_Y + 1) AND BYTE#16#0F) OR BYTE#16#30;

		in_Write_Index := in_Write_Index + INT#1;
		S_BUF.BUFFER[in_Write_Index] := BYTE#16#3B; (* ; *)

		(* output tens digit of column number *)
		in_Write_Index := in_Write_Index + INT#1;
		S_BUF.BUFFER[in_Write_Index] := SHR(INT_TO_BCDC(Xus_TN_SCREEN.in_Cursor_X + 1),INT#4) OR BYTE#16#30;

		(* output ones digit of column number *)
		in_Write_Index := in_Write_Index + INT#1;
		S_BUF.BUFFER[in_Write_Index] := (INT_TO_BCDC(Xus_TN_SCREEN.in_Cursor_X + 1) AND BYTE#16#0F) OR BYTE#16#30;

		in_Write_Index := in_Write_Index + INT#1;
		S_BUF.BUFFER[in_Write_Index] := BYTE#16#48; (* H *)

END_IF;

(* store current write index -> trigger send *)
S_BUF.SIZE := INT_TO_UINT(in_Write_Index + 1);
END_FUNCTION_BLOCK

// Commented out for beedance: it reads or writes the bytes of a STRING through a pointer; a beedance reference (REF_TO) refers to a whole variable of its type.
// FUNCTION_BLOCK UNI_CIRCULAR_BUFFER
// VAR_IN_OUT
// 	DATA : UNI_CIRCULAR_BUFFER_DATA;
// END_VAR
// VAR_TEMP
// 	tmp_dw : DWORD;
// 	pTmp : REF_TO BYTE;
// 	n : INT;
// 	n1 : INT;
// 	n2 : INT;
// 	x: BYTE;
// 	buf_totalsize : UINT;
// END_VAR
// VAR CONSTANT
// 	HeaderSize : INT := 4;
// END_VAR
// VAR
// 	cnt : UINT;
// 	mode_last : INT;
//
// 	(*LOG_MSG : LOG_MSG;
// 	_debug_enable : BOOL := FALSE;*)
// END_VAR
//
// CASE DATA.D_MODE OF
//
// 01:	x := WORD_TO_BYTE(DATA.D_HEAD); (* evaluate only the right byte *)
// 	CASE x OF
// 	01:	cnt := LEN(DATA.D_STRING); (* process string *)
// 		pTmp := REF(DATA.D_STRING);
// 	02:	cnt := 4; (* process real *)
// 		pTmp := REF(DATA.D_REAL);
// 	03:	cnt := 4; (* process DWORD *)
// 		pTmp := REF(DATA.D_DWORD);
// 	ELSE
// 		cnt := 0;
// 	END_CASE;
//
// 	DATA.BUF_DATA_CNT := DATA.BUF_DATA_CNT + UDINT#1;
//
// 	(* ------ enter data into buffer ------ *)
// 	buf_totalsize := SIZEOF(DATA.BUF);
//
// 	IF (cnt + HeaderSize) > (buf_totalsize - DATA.BUF_SIZE) THEN (* enough memory free? *)
// 		DATA.BUF_DATA_LOST := DATA.BUF_DATA_LOST + UDINT#1;
// 		RETURN;
// 	END_IF;
//
// 	DATA.D_SIZE := cnt;
//
// 	mode_last := DATA.D_MODE;
// 	tmp_dw := SHL(WORD_TO_DWORD(DATA.D_HEAD),16) OR UINT_TO_DWORD(cnt);
//
// 	(* enter header into buffer *)
// 	n1 := 0;
// 	REPEAT
// 		n2 := MIN(HeaderSize - n1, buf_totalsize - DATA._Last);
// 		FOR n := 1 TO n2 DO
// 			tmp_dw := ROL(tmp_dw,8);
// 			data.BUF[DATA._Last] := DWORD_TO_BYTE(tmp_dw);
// 			DATA._Last := DATA._Last + 1;
// 		END_FOR;
// 		IF DATA._Last >= buf_totalsize THEN
// 			DATA._Last := 0;
// 		END_IF
// 		n1 := n1 + n2;
// 	UNTIL n1 >= HeaderSize
// 	END_REPEAT;
//
// 	(* enter data into buffer *)
// 	n1 := 0;
// 	REPEAT
// 		n2 := MIN(cnt - n1, buf_totalsize - DATA._Last);
// 		FOR n := 1 TO n2 DO
// 			data.BUF[DATA._Last] := pTmp^;
// 			pTmp := pTmp + 1;
// 			DATA._Last := DATA._Last + 1;
// 		END_FOR;
// 		IF DATA._Last >= buf_totalsize THEN
// 			DATA._Last := 0;
// 		END_IF
// 		n1 := n1 + n2;
// 	UNTIL n1 >= cnt
// 	END_REPEAT;
//
// 	DATA.BUF_SIZE := DATA.BUF_SIZE + cnt + HeaderSize;
// 	DATA.BUF_COUNT := DATA.BUF_COUNT + 1;
// 	DATA.BUF_USED := UINT_TO_USINT(100 * DATA.BUF_SIZE / buf_totalsize); (* used memory in % *)
// 	DATA.D_MODE := 0;
//
// 	(*####################  DEBUG-MESSAGE  ###################################*)
// 	(*IF _debug_enable THEN
// 		LOG_CL.NEW_MSG := 'RP: ADD /HEAD ~1 / SIZE ~2 / CNT ~3 / >~4<';
// 		LOG_CL.PRINTF[1] := DWORD_TO_STRH(DATA.D_HEAD);
// 		LOG_CL.PRINTF[2] := UINT_TO_STRING(cnt);
// 		LOG_CL.PRINTF[3] := UINT_TO_STRING(DATA.BUF_COUNT);
// 		CASE x OF
// 		01:	LOG_CL.PRINTF[4] := DATA.D_STRING;
// 		02:	LOG_CL.PRINTF[4] := REAL_TO_STRING(DATA.D_REAL);
// 		03:	LOG_CL.PRINTF[4] := DWORD_TO_STRH(DATA.D_DWORD);
// 		ELSE
// 			LOG_CL.PRINTF[4] := '';
// 		END_CASE;
// 		LOG_MSG();
// 	END_IF;*)
// 	(*########################################################################*)
//
// 10..12:	(* ------ read data from buffer and optionally delete ------ *)
// 		(* 10 = read only / 11 = delete after read / 12 = read and delete *)
// 	IF DATA.D_MODE <> 11 THEN
// 		IF DATA.BUF_COUNT = 0 THEN RETURN; END_IF;
// 		buf_totalsize := SIZEOF(DATA.BUF);
// 		DATA._GetEnd := DATA._First;(* remember index of the oldest entry *)
// 		mode_last := DATA.D_MODE;
//
// 		(* read header from buffer *)
// 		n1 := 0;
// 		tmp_dw := 0;
// 		REPEAT
// 			n2 := MIN(HeaderSize - n1, buf_totalsize - DATA._GetEnd);
// 			FOR n := 1 TO n2 DO
// 				tmp_dw := ROL(tmp_dw,8) OR BYTE_TO_DWORD(data.BUF[DATA._GetEnd]);
// 				DATA._GetEnd := DATA._GetEnd + 1;
// 			END_FOR;
// 			IF DATA._GetEnd >= buf_totalsize THEN
// 				DATA._GetEnd := 0;
// 			END_IF
// 			n1 := n1 + n2;
// 		UNTIL n1 >= HeaderSize
// 		END_REPEAT;
//
// 		DATA._GetStart := DATA._GetEnd;
// 		cnt := DWORD_TO_UINT(tmp_dw AND 16#0000_FFFF);
// 		DATA.D_SIZE := cnt;
// 		DATA.D_HEAD := DWORD_TO_WORD(SHR(tmp_dw,16));
//
// 		x := WORD_TO_BYTE(DATA.D_HEAD); (* evaluate only the right byte *)
// 		CASE x OF
// 		01:	pTmp := REF(DATA.D_STRING); (* process string *)
// 		02:	pTmp := REF(DATA.D_REAL); (* process real *)
// 		03:	pTmp := REF(DATA.D_DWORD); (* process DWORD *)
// 		END_CASE;
//
// 		(* read data from buffer *)
// 		n1 := 0;
// 		REPEAT
// 			n2 := MIN(cnt - n1, buf_totalsize - DATA._GetEnd);
// 			FOR n := 1 TO n2 DO
// 				pTmp^ := data.BUF[DATA._GetEnd];
// 				pTmp := pTmp + 1;
// 				DATA._GetEnd := DATA._GetEnd + 1;
// 			END_FOR;
// 			IF DATA._GetEnd >= buf_totalsize THEN
// 				DATA._GetEnd := 0;
// 			END_IF
// 			n1 := n1 + n2;
// 		UNTIL n1 >= cnt
// 		END_REPEAT;
// 		IF x = 1 THEN
// 			pTmp^ := 0; (* terminate string *)
// 		END_IF;
// 		DATA.D_MODE := 0;
//
// 		(*####################  DEBUG-MESSAGE  ###################################*)
// 		(*IF _debug_enable THEN
// 			LOG_CL.NEW_MSG := 'RP: READ /HEAD ~1 / SIZE ~2 / CNT ~3 / >~4<';
// 			LOG_CL.PRINTF[1] := DWORD_TO_STRH(DATA.D_HEAD);
// 			LOG_CL.PRINTF[2] := UINT_TO_STRING(cnt);
// 			LOG_CL.PRINTF[3] := UINT_TO_STRING(DATA.BUF_COUNT);
// 			CASE x OF
// 			01:	LOG_CL.PRINTF[4] := DATA.D_STRING;
// 			02:	LOG_CL.PRINTF[4] := REAL_TO_STRING(DATA.D_REAL);
// 			03:	LOG_CL.PRINTF[4] := DWORD_TO_STRH(DATA.D_DWORD);
// 			ELSE
// 				LOG_CL.PRINTF[4] := '';
// 			END_CASE;
// 			LOG_MSG();
// 		END_IF;*)
// 		(*########################################################################*)
// 	END_IF;
//
// 	IF (mode_last = 10 AND DATA.D_MODE = 11) OR (mode_last = 12 AND DATA.D_MODE = 0) THEN (* delete only possible directly after read *)
// 		mode_last := DATA.D_MODE;
// 		DATA.BUF_SIZE := DATA.BUF_SIZE - cnt - HeaderSize;
// 		DATA.BUF_COUNT := DATA.BUF_COUNT - 1;
// 		DATA._First := DATA._GetEnd;
// 		DATA.BUF_USED := UINT_TO_USINT(100 * DATA.BUF_SIZE / SIZEOF(DATA.BUF)); (* used memory in % *)
// 		DATA.D_MODE := 0;
//
// 		(*####################  DEBUG-MESSAGE  ###################################*)
// 		(*IF _debug_enable THEN
// 			LOG_CL.NEW_MSG := 'RP: DEL /HEAD ~1 / SIZE ~2 / CNT ~3 / >~4<';
// 			LOG_CL.PRINTF[1] := DWORD_TO_STRH(DATA.D_HEAD);
// 			LOG_CL.PRINTF[2] := UINT_TO_STRING(cnt);
// 			LOG_CL.PRINTF[3] := UINT_TO_STRING(DATA.BUF_COUNT);
// 			CASE x OF
// 			01:	LOG_CL.PRINTF[4] := DATA.D_STRING;
// 			02:	LOG_CL.PRINTF[4] := REAL_TO_STRING(DATA.D_REAL);
// 			03:	LOG_CL.PRINTF[4] := DWORD_TO_STRH(DATA.D_DWORD);
// 			ELSE
// 				LOG_CL.PRINTF[4] := '';
// 			END_CASE;
// 			LOG_MSG();
// 		END_IF;*)
// 		(*########################################################################*)
// 	END_IF;
//
// 99:	(* buffer reset - delete everything *)
// 	DATA._First := 0;
// 	DATA._Last := 0;
// 	DATA._GetStart := 0;
// 	DATA._GetEnd := 0;
// 	DATA.BUF_COUNT := 0;
// 	DATA.BUF_SIZE := 0;
// 	DATA.BUF_USED := 0;
// 	DATA.D_STRING := '';
// 	DATA.D_DWORD := 0;
// 	DATA.D_REAL := 0.0;
// 	DATA.D_HEAD := 0;
// 	DATA.D_MODE := 0;
// 	DATA.D_SIZE := 0;
// 	mode_last := 0;
// END_CASE;
//
// (* store highest utilization value *)
// IF DATA.BUF_USED > DATA.BUF_USED_MAX THEN
// 	DATA.BUF_USED_MAX := DATA.BUF_USED;
// END_IF;
// END_FUNCTION_BLOCK

// Commented out for beedance: it uses CHR_TO_STRING, which is commented out.
// FUNCTION URL_DECODE : STRING(STRING_LENGTH)
// VAR_INPUT
// 	IN : STRING(STRING_LENGTH);
// END_VAR
// VAR
// 	pos : INT;
// 	seq : STRING(3);
// 	new : STRING(1);
// END_VAR
//
// URL_DECODE := IN;
// pos := FIND(URL_DECODE,'%');
// WHILE pos > 0 DO
// 	seq := MID(URL_DECODE,2,pos + 1);
// 	new := CHR_TO_STRING(DWORD_TO_BYTE(HEX_TO_DWORD(seq)));
// 	URL_DECODE := REPLACE(URL_DECODE, new, 3, pos);
// 	pos := FIND(URL_DECODE,'%');
// END_WHILE;
// END_FUNCTION

// Commented out for beedance: it reads or writes the bytes of a STRING through a pointer; a beedance reference (REF_TO) refers to a whole variable of its type.
// FUNCTION URL_ENCODE : STRING(STRING_LENGTH)
// VAR_INPUT
// 	IN : STRING(STRING_LENGTH);
// END_VAR
// VAR
// 	pt_in : REF_TO ARRAY[1..255] OF BYTE;
// 	pt_out : REF_TO ARRAY[1..256] OF BYTE;
// 	pos_in : INT;
// 	pos_out : INT;
// 	stop : INT;
// 	tb : BYTE;
// END_VAR
//
// pt_in  := REF(in);
// pt_out := REF(URL_ENCODE);
//
// (* scan the input string and convert unallowed characters *)
// pos_in := 1;
// stop := LEN(in);
// FOR pos_out := 1 TO 250 DO
// 	IF pos_in > stop THEN
// 		EXIT;
// 	ELSIF IS_URLCHR(pt_in^[pos_in]) THEN
// 		pt_out^[pos_out] := pt_in^[pos_in];
// 		(* increment in by 1 *)
// 		pos_in := pos_in + 1;
// 	ELSE
// 		(* cannot fit 3 digits, exit *)
// 		IF pos_out > 248 THEN EXIT; END_IF;
// 		(* invalid character that needs to be converted *)
// 		pt_out^[pos_out] := 37;    (* start with % sign *)
// 		pos_out := pos_out + 1;
// 		(* need to add the two hex digits *)
// 		tb := SHR(pt_in^[pos_in],4);
// 		IF tb > 9 THEN
// 			pt_out^[pos_out] := tb + 55;
// 		ELSE
// 			pt_out^[pos_out] := tb + 48;
// 		END_IF;
// 		pos_out := pos_out + 1;
// 		tb := pt_in^[pos_in] AND 16#0F;
// 		IF tb > 9 THEN
// 			pt_out^[pos_out] := tb + 55;
// 		ELSE
// 			pt_out^[pos_out] := tb + 48;
// 		END_IF;
// 		(* increment in and out because out has to move 3 digits *)
// 		pos_in := pos_in + 1;
// 	END_IF;
// END_FOR;
//
// (* terminate the output string *)
// pt_out^[pos_out] := 0;
// END_FUNCTION

FUNCTION URL_TO_STRING : STRING(STRING_LENGTH)
VAR_INPUT
	IN : URL;
END_VAR

(* attach protocol *)
IF IN.PROTOCOL <> '' THEN URL_TO_STRING := CONCAT(IN.PROTOCOL,'://'); END_IF;

(* attach user and password *)
IF IN.USER <> '' THEN
	URL_TO_STRING := CONCAT(URL_TO_STRING, IN.USER);
	IF IN.PASSWORD <> '' THEN
		URL_TO_STRING := CONCAT(URL_TO_STRING, ':');
		URL_TO_STRING := CONCAT(URL_TO_STRING, IN.PASSWORD);
	END_IF;
	URL_TO_STRING := CONCAT(URL_TO_STRING, '@');
END_IF;

(* attach domain *)
URL_TO_STRING := CONCAT(URL_TO_STRING, IN.DOMAIN);

(* attach Port *)
IF IN.PORT > 0 THEN
	URL_TO_STRING := CONCAT(URL_TO_STRING, ':');
	URL_TO_STRING := CONCAT(URL_TO_STRING, WORD_TO_STRING(IN.PORT));
END_IF;

(* attach path *)
URL_TO_STRING := CONCAT(URL_TO_STRING, IN.PATH);

(* attach query *)
IF IN.QUERY <> '' THEN
	URL_TO_STRING := CONCAT(URL_TO_STRING, '?');
	URL_TO_STRING := CONCAT(URL_TO_STRING, IN.QUERY);
END_IF;

(* attach anchor *)
IF IN.ANCHOR <> '' THEN
	URL_TO_STRING := CONCAT(URL_TO_STRING, '#');
	URL_TO_STRING := CONCAT(URL_TO_STRING, IN.ANCHOR);
END_IF;
END_FUNCTION

// Commented out for beedance: it uses CSV_PARSER_BUF, which is commented out.
// FUNCTION_BLOCK WORLD_WEATHER
// VAR_IN_OUT
// 	IP_C : IP_C; (* IP_Control management structure *)
// 	S_BUF : NETWORK_BUFFER;
// 	R_BUF : NETWORK_BUFFER;
// 	WW : WORLD_WEATHER_DATA;
// END_VAR
// VAR_INPUT
// 	ACTIVATE : BOOL;
// 	LATITUDE : REAL;
// 	LONGITUDE : REAL;
// 	KEY : STRING(30);
// END_VAR
// VAR_OUTPUT
// 	BUSY : BOOL;
// 	DONE : BOOL;
// 	ERROR_C : DWORD;
// 	ERROR_T : BYTE;
// END_VAR
// VAR
// 	URL_DATA : url;
// 	DNS_CLIENT : DNS_CLIENT;
// 	HTTP_GET : HTTP_GET;
// 	CPB : CSV_PARSER_BUF;
// 	last_state : BOOL;
// 	value_int : INT;
// 	value_real : REAL;
// 	v_real : REAL;
// 	state : INT;
// 	url_str : STRING(STRING_LENGTH);
// 	offset : UDINT;
// 	size : INT;
// 	sep : BYTE;
// 	cnt : INT;
// 	day : INT;
// 	idx : INT;
// 	run : BYTE;
// 	result : BYTE;
// 	value : STRING(STRING_LENGTH);
// 	pos : INT;
// END_VAR
//
// CASE state OF
//
// 00:
// 	IF ACTIVATE AND NOT last_state THEN
// 		state := 20;
// 		DONE := FALSE;
// 		BUSY := TRUE;
// 		ERROR_C := DWORD#0;
// 		ERROR_T := BYTE#0;
// 	END_IF;
//
// 20: (* URL for DNS AND HTTP-GET *)
// 	(* Example: http://api.worldweatheronline.com/free/v1/weather.ashx?q=48.21,16.37&format=csv&num_of_days=5&key=xxxxxxxxxxxxxxxxxxxxxx *)
// 	url_str := CONCAT('http://api.worldweatheronline.com/free/v1/weather.ashx?q=',REAL_TO_STRF(LATITUDE,6,D:='.'));
// 	url_str := CONCAT(url_str,',');
// 	url_str := CONCAT(url_str,REAL_TO_STRF(LONGITUDE,6,D:='.'));
// 	url_str := CONCAT(url_str,'&format=csv&num_of_days=5&key=');
// 	url_str := CONCAT(url_str,key);
//
// 	URL_DATA:=STRING_TO_URL(STR:=url_str, DEFAULT_PROTOCOL:='', DEFAULT_PATH:='' );
// 	state := 40;
//
// 40:
// 	IF DNS_CLIENT.DONE THEN
// 		state := 60;
// 	ELSIF (DNS_CLIENT.ERROR > DWORD#00) THEN
// 		(* error handling *)
// 		ERROR_C := DNS_CLIENT.ERROR;
// 	ERROR_T := BYTE#01;
// 		state   := 100;
// 	END_IF;
//
// 60:
// 	IF HTTP_GET.DONE THEN
// 		sep := 0;
// 		idx := 0;
// 		day := 0;
// 		cnt := 0;
// 		OFFSET := HTTP_GET.BODY_START; (* set start offset *)
// 		size := HTTP_GET.BODY_STOP; (* End Position *)
// 		run := 1; (* search element *)
// 		state := 80;
//
// 	ELSIF (HTTP_GET.ERROR > DWORD#00) THEN
// 		(* error handling *)
// 		ERROR_C := HTTP_GET.ERROR;
// 		ERROR_T := BYTE#02;
// 		state := 100;
// 	END_IF;
//
// 80:	IF run = 0 THEN (* no command active anymore? *)
// 		run := 1; (*  search next element  *)
// 		IF result = 1 OR result = 2 THEN
// 			value_int := 0;
// 			value_real := 0.0;
// 			(* perform automatic conversion to real and int *)
// 			IF LEN(value) <= 20 THEN
// 				v_real:=FLOAT_TO_REAL(FLT:=value);
// 				IF CHK_REAL(v_real) = 0 THEN (* !!! checks for a valid REAL value, otherwise TwinCAT crashes !!!!  *)
// 					value_real := v_real;
// 					value_int := REAL_TO_INT(value_real);
// 				END_IF;
// 			END_IF;
// 			cnt := cnt + 1;
//
// 			IF cnt = 1 AND LEFT(value,1) <> '#' THEN
// 				cnt := 0;
// 			END_IF;
//
// 			IF cnt >=8 AND cnt <= 87 THEN
// 				IF cnt > 22 THEN
// 					CASE idx OF
// 					00:	WW.DAY[day].DATE_OF_DAY := value;
// 					01:	WW.DAY[day].TEMP_MAX_C := value_int;
// 					02:	WW.DAY[day].TEMP_MAX_F := value_int;
// 					03:	WW.DAY[day].TEMP_MIN_C := value_int;
// 					04:	WW.DAY[day].TEMP_MIN_F := value_int;
// 					05:	WW.DAY[day].WIND_SPEED_MILES := value_int;
// 					06:	WW.DAY[day].WIND_SPEED_KMPH := value_int;
// 					07:	WW.DAY[day].WIND_DIR_DEGREE := value_int;
// 					08:	WW.DAY[day].WIND_DIR16POINT := value;
// 					09:	WW.DAY[day].WEATHER_CODE := value_int;
// 					10:	pos := FIND(value, '/wsymbol_');
// 						WW.DAY[day].WEATHER_ICON := DEC_TO_INT(MID(value,4,pos+9));
// 					11:	WW.DAY[day].WEATHER_DESC := value;
// 					12:	WW.DAY[day].PRECIPMM := value_real;
// 					END_CASE;
// 					idx := idx + 1;
// 					IF idx > 12 THEN
// 						idx := 0;
// 						day := day + 1;
// 					END_IF;
// 				ELSE
// 					CASE cnt OF
// 					08:	sep :=44; (* from now on work with separators, *)
// 					09:	WW.CUR.OBSERVATION_TIME := value;
// 					10:	WW.CUR.TEMP_C := value_int;
// 					11:	WW.CUR.WEATHER_CODE := value_int;
// 					12:	pos := FIND(value, '/wsymbol_');
// 						WW.CUR.WEATHER_ICON := DEC_TO_INT(MID(value,4,pos+9));
// 					13:	WW.CUR.WEATHER_DESC := value;
// 					14:	WW.CUR.WIND_SPEED_MILES := value_int;
// 					15:	WW.CUR.WIND_SPEED_KMPH := value_int;
// 					16:	WW.CUR.WIND_DIR_DEGREE := value_int;
// 					17:	WW.CUR.WIND_DIR16POINT := value;
// 					18:	WW.CUR.PRECIPMM := value_real;
// 					19:	WW.CUR.HUMIDITY := value_int;
// 					20:	WW.CUR.VISIBILITY := value_int;
// 					21:	WW.CUR.PRESSURE := value_int;
// 					22:	WW.CUR.CLOUDOVER := value_int;
// 					END_CASE;
// 				END_IF;
// 			END_IF;
// 		ELSIF result = 10 THEN (* nothing more found *)
// 			DONE  := TRUE;
// 			run := 0; (* end evaluation *)
// 			state := 100;
// 		END_IF;
// 	END_IF;
//
// 100:
// 	(* UNLOCK HTTP DATA *)
// 	IF (NOT HTTP_GET.DONE) THEN
// 		state := 0;
// 		BUSY := FALSE;
// 		DONE := ERROR_T = BYTE#0;
// 	END_IF;
//
// END_CASE;
//
// (* ---------------- DNS --------------- *)
// DNS_CLIENT(	IP_C:=IP_C,
// 			S_BUF:=S_BUF,
// 			R_BUF:=R_BUF,
// 			DOMAIN:=URL_DATA.DOMAIN,
// 			IP4_DNS:=DWORD#00,
// 			ACTIVATE:=state=40 (* DNS Start *)
// 			);
// (* parameters not used, or not used directly *)
// (*	DWORD :=DNS_CLIENT.IP4;
// 	BOOL  :=DNS_CLIENT.DONE;
// 	BYTE  :=DNS_CLIENT.ERROR; *)
// (* -------------------------------------*)
//
// (* ------------- HTTP_GET --------------- *)
// HTTP_GET(	IP_C:=IP_C,
// 			S_BUF:=S_BUF,
// 			R_BUF:=R_BUF,
// 			IP4:=DNS_CLIENT.IP4,
// 			GET:=state=60,
// 			MODE:=BYTE#2, (* HTTP 1.1 with persistent connection *)
// 			UNLOCK_BUF:=state=100,
// 			URL_DATA:=URL_DATA
// 			);
//
// (* parameters not used, or not used directly *)
// (*	STRING := HTTP_GET.HTTP_STATUS;
// 	UINT :=HTTP_GET.HEADER_START;
// 	UINT :=HTTP_GET.HEADER_STOP;
// 	UINT :=HTTP_GET.BODY_START;
// 	UINT :=HTTP_GET.BODY_STOP;
// 	BOOL :=HTTP_GET.DONE;
// 	BYTE :=HTTP_GET.ERROR;
// *)
// (* -------------------------------------*)
// CPB(SEP:=sep,RUN:=run,OFFSET:=OFFSET,VALUE:=value,PT:=R_BUF,RESULT=>result); (* CSV PARAMETER BUF *)
//
// last_state := ACTIVATE;
// END_FUNCTION_BLOCK

FUNCTION_BLOCK WORLD_WEATHER_DESC_GE
VAR_IN_OUT
	WW : WORLD_WEATHER_DATA;
END_VAR
VAR_INPUT
	ACTIVATE : BOOL;
END_VAR
VAR
	act_last : BOOL;
	x : INT;
	y : INT;
	str : STRING(60);
	i : INT;
END_VAR

IF ACTIVATE AND act_last = FALSE THEN
	i := 0;
	FOR y := 1 TO 12 DO
		CASE y OF
		1,3,5,7,9:		x :=  WW.DAY[i].WEATHER_CODE;
		2,4,6,8,10:	WW.DAY[i].WEATHER_DESC := str;
					i := i + 1;
		11:			x :=  WW.CUR.WEATHER_CODE;
		12:			WW.CUR.WEATHER_DESC := str;
		END_CASE;

		CASE x OF
			113	:	str := 'heiter/sonnig';
			116	:	str := 'stellenweise wolkig';
			119	:	str := 'wolkig';
			122	:	str := 'bewölkt';
			143	:	str := 'Nebel';
			176	:	str := 'stellenweise nahegelegener Regen';
			179	:	str := 'stellenweise nahegelegener Schneefall';
			182	:	str := 'stellenweise nahegelegener Eisregen';
			185	:	str := 'stellenweise gefrierender Niesel';
			200	:	str := 'nahegelegene Sturm';
			227	:	str := 'Schneetreiben';
			230	:	str := 'Schneesturm';
			248	:	str := 'Nebel';
			260	:	str := 'gefrierender Nebel';
			263	:	str := 'stellenweise leichter Nieselregen';
			266	:	str := 'leichter Niesel';
			281	:	str := 'gefrierender Nieselregen';
			284	:	str := 'stark gefrierender Nieselregen';
			293	:	str := 'stellenweise leichter Regen';
			296	:	str := 'leichter Regen';
			299	:	str := 'zeitweise etwas Regen';
			302	:	str := 'mäßiger Regen';
			305	:	str := 'zeitweise etwas starker Regen';
			308	:	str := 'starker Regen';
			311	:	str := 'leichter gefrierender Regen';
			314	:	str := 'mäßiger oder starker Eisregen';
			317	:	str := 'leichter Eisregen';
			320	:	str := 'mäßiger oder starker Eisregen';
			323	:	str := 'stellenweise leichter Schneefall';
			326	:	str := 'leichter Scheefall';
			329	:	str := 'stellenweise moderater Schneefall';
			332	:	str := 'mäßiger Schnee';
			335	:	str := 'stellenweise starker Scheefall';
			338	:	str := 'starker Schneefall';
			350	:	str := 'Hagel';
			353	:	str := 'leichte Regenfälle';
			356	:	str := 'mäßiger oder starker Regenfall';
			359	:	str := 'sintflutartige Regenfälle';
			362	:	str := 'leichter Eisregen';
			365	:	str := 'mäßiger oder starker Eisregen';
			368	:	str := 'leichte Schneeschauer';
			371	:	str := 'mäßiger oder starker Schneefall';
			374	:	str := 'leichter Hagel';
			377	:	str := 'mäßiger oder starker Hagel';
			386	:	str := 'stellenweise leichter Regen in Gewittergebiet';
			389	:	str := 'mäßiger oder starker Regen in Gewittergebiet';
			392	:	str := 'stellenweise leichter Schneefall in Gewittergebiet';
			395	:	str := 'mäßiger oder starker Schnee in Gewittergebiet';
		ELSE
			str := 	'nicht verfügbar';
		END_CASE;
	END_FOR;
END_IF;
act_last := ACTIVATE;
END_FUNCTION_BLOCK

FUNCTION_BLOCK WORLD_WEATHER_ICON_OSCAT
VAR_IN_OUT
	WW : WORLD_WEATHER_DATA;
END_VAR
VAR_INPUT
	ACTIVATE : BOOL;
END_VAR
VAR
	dat : ARRAY[0..41] OF INT := 0,14,12,9,9,0,7,7,0,2,2,3,3,1,0,0,17,4,4,3,3,1,0,0,17,2,2,3,3,1,0,0,17,2,4,3,3,1,0,0,17,0;
	act_last : BOOL;
	x : INT;
	i : INT;
END_VAR

IF ACTIVATE AND act_last = FALSE THEN
	x := LIMIT(0,WW.CUR.WEATHER_ICON,41);
	WW.CUR.WEATHER_ICON := dat[x];
	FOR i := 0 TO 4 DO
		x := LIMIT(0,WW.DAY[i].WEATHER_ICON,41);
		WW.DAY[i].WEATHER_ICON := dat[x];
	END_FOR;
END_IF;
act_last := ACTIVATE;
END_FUNCTION_BLOCK

// Commented out for beedance: it uses BUFFER_TO_STRING, which is commented out.
// FUNCTION_BLOCK XML_READER
// VAR_IN_OUT
// 	CTRL : XML_CONTROL;
// 	BUF : NW_BUF_LONG;
// END_VAR
// VAR
// 	index :	INT;
// 	index2 : INT;
// 	stop : INT;
// 	mode : INT;
// 	command : WORD;
// 	c :	BYTE;
// 	s1 : INT;
// 	e1 : INT;
// 	path_overflow : BOOL;
// 	empty_tag : BOOL;
// 	s_code : STRING(10);
// 	e_code : STRING(10);
// 	watchdog : TON;
//
// 	(*LOG_MSG : LOG_MSG;
// 	_debug_enable : BOOL := TRUE;*)
//
// END_VAR
//
// (*
//
// TYP
// 00 = UNKNOWN
// 01 = ELEMENT (STANDARD)
// 02 = CLOSE ELEMENT
// 03 = TEXT
// 04 = ATTRIBUTE
// 05 = ELEMENT (PROCESSING INSTRUCTION)
//
// 12 = !CDATA
// 13 = !COMMENT
// 14 = !DTD ELEMENT (Document Type Declarations )
//
// 98 = WATCHDOG
// 99 = END
//
// no block data is output for type 02!
//
// *)
//
// (* ---------- Init -------------- *)
// IF BIT_OF_DWORD(WORD_TO_DWORD(CTRL.COMMAND),15) THEN
// 	COMMAND := CTRL.COMMAND;
// 	CTRL.COMMAND := WORD#0;
//
// 	index := UINT_TO_INT(CTRL.START_POS);
// 	stop := UINT_TO_INT(CTRL.STOP_POS);
// 	mode := 100;
// 	path_overflow := FALSE;
//
// 	CTRL.TYP := 0;
// 	CTRL.COUNT := UINT#00;
// 	CTRL.LEVEL := UINT#00;
// 	CTRL.ATTRIBUTE := '';
// 	CTRL.ELEMENT := '';
// 	CTRL.PATH := '';
// 	CTRL.VALUE := '';
//
// 	WATCHDOG.PT := CTRL.WATCHDOG;
// END_IF;
//
// (*----------------------------------------------- *)
//
// IF index < 0 THEN RETURN;END_IF;
//
// CTRL.BLOCK1_START := UINT#0;
// CTRL.BLOCK1_STOP := UINT#0;
// CTRL.BLOCK2_START := UINT#0;
// CTRL.BLOCK2_STOP := UINT#0;
//
// WATCHDOG(IN:=FALSE); (* stop timer *)
//
// WHILE (TRUE) DO
//
// 	(* -------------- WATCHDOG ------------------ *)
// 	WATCHDOG(IN:=CTRL.WATCHDOG > T#0s);
// 	IF WATCHDOG.Q THEN
// 		CTRL.TYP := 98;
//     		(*####################  DEBUG-MESSAGE  ###################################*)
//     		(*IF _debug_enable THEN
//       			LOG_CL.NEW_MSG := 'WATCHDOG:';
//       			LOG_MSG();
//     		END_IF;*)
//     		(*########################################################################*)
// 		RETURN;
// 	END_IF;
//
// 	(* -------------- PARSING END ------------------ *)
// 	IF index > stop THEN
// 		CTRL.COUNT := CTRL.COUNT + UINT#1;
// 		CTRL.TYP := 99;
//     		(*####################  DEBUG-MESSAGE  ###################################*)
//     		(*IF _debug_enable THEN
//       			LOG_CL.NEW_MSG := 'EX: #T:~1 #C:~2 #P:~6 #L:~7';
//       			LOG_CL.PRINTF[1] := INT_TO_STRING(CTRL.TYP);
//       			LOG_CL.PRINTF[2] := UINT_TO_STRING(CTRL.COUNT);
//       			LOG_CL.PRINTF[6] := CTRL.PATH;
//       			LOG_CL.PRINTF[7] := UINT_TO_STRING(CTRL.LEVEL);
//       			LOG_MSG();
//     		END_IF;*)
//     		(*########################################################################*)
// 		mode  := 0; (* reset step *)
// 		index := 0; (* stop processing *)
// 		RETURN;
// 	END_IF;
//
// 	CASE mode OF
//
// 	100: (* ---------- ELEMENT SECTION ------------------ *)
// 		(* search begin of element *)
// 		s1 := 0;
// 		e1 := 0;
// 		WHILE (index <= stop) DO
// 			IF BUF[INDEX]=BYTE#60 THEN (* '<' TagBegin *)
// 				index := index + 1;
// 				C := BUF[index];
// 				IF C = BYTE#47 THEN (* '/' TagTerm *)
// 					mode := 300; (* End Element Section *)
// 				ELSIF C = BYTE#33 THEN (* '!' for Special Section *)
// 					index := index + 1;
// 					mode := 500;
// 				ELSE
// 					s1 := index;
// 				END_IF;
// 				EXIT;
// 			END_IF;
// 			index := index + 1;
// 		END_WHILE;
//
// 		(* analyse element *)
// 		CTRL.TYP := 0; (* clear TYPE *)
// 		IF s1 > 0 THEN
// 			WHILE (index <= stop AND e1 = 0) DO
// 				c := BUF[index];
// 				(* whitespace character = element with attributes *)
// 				IF c <= BYTE#32 THEN
// 					(* search next printable character *)
// 					index2 := index;
// 					WHILE (index2 <= stop) AND (BUF[index2] <= BYTE#32) DO
// 						index2 := index2 + 1;
// 					END_WHILE;
// 					IF BUF[index2] = BYTE#47 THEN (* check for empty element '/' *)
// 						index := index2;
// 						e1 := index - 2;
// 						CTRL.TYP := 1; (* structure element *)
// 						mode := 300;   (* Close Element *)
// 						EXIT;
// 					END_IF;
//
// 					e1 := index - 1;
// 					CTRL.TYP := 1; (* element with attributes *)
// 					mode := 400;
//
// 				ELSIF c = BYTE#62 THEN (* '>' TagEnd *)
//
// 					(* check for empty element <xx/> *)
// 					index2 := index - 1;
// 					IF BUF[index2] = BYTE#47 THEN (* TagTerm '/' *)
// 						e1 := index2 - 1;
// 						CTRL.TYP := 1;
// 						EMPTY_TAG := TRUE; (* EMPTY TAG Mode *)
// 						mode := 200; (* TEXT Element *)
// 						EXIT;
// 					END_IF;
//
// 					e1 := index - 1;
// 					index2 := index + 1;
//
// 					(* examine following element *)
// 					WHILE (index2 <= stop) DO
// 						c := BUF[index2];
// 						IF c = BYTE#60 THEN (* '<' TagBegin *)
//
// 							index2 := index2 + 1; (* unfortunately no other way on PCWORX!*)
// 							c := BUF[index2];
// 							index2 := index2 - 1;
// 							IF c = BYTE#47 THEN (* TagTerm '/' *)
// 								empty_tag := TRUE;
// 								mode := 200; (* TEXT Element *)
// 							ELSE
// 								mode := 100; (* Element *)
// 							END_IF;
// 							CTRL.TYP := 1; (* structure element *)
// 							EXIT;
// 						ELSIF c > BYTE#32  THEN (* Printable-Character *)
// 							CTRL.TYP := 1; (* element with text *)
// 							mode := 200;
// 							EXIT;
// 						END_IF;
// 						index2 := index2 + 1;
// 					END_WHILE;
// 				END_IF;
// 				index := index + 1;
// 			END_WHILE;
// 		END_IF;
//
// 		(* new element found*)
// 		IF CTRL.TYP > 0 THEN
//
// 			(* special check for processing instruction (PI) *)
// 			IF BUF[s1] = BYTE#63 THEN (* '?' for Processing Instruction *)
// 				s1 := s1 + 1; (* skip leading '?' *)
// 				CTRL.TYP := 5;
// 			END_IF;
// 			CTRL.BLOCK1_START := INT_TO_UINT(s1);
// 			CTRL.BLOCK1_STOP  := INT_TO_UINT(e1);
// 			CTRL.ELEMENT := BUFFER_TO_STRING(PT:=REF(BUF),SIZE:=INT_TO_UINT(stop + 1),START:=CTRL.BLOCK1_START,STOP:=CTRL.BLOCK1_STOP);
// 			CTRL.COUNT := CTRL.COUNT + UINT#1;
// 			CTRL.LEVEL := CTRL.LEVEL + UINT#1;
//
// 			IF path_overflow = FALSE THEN
// 				(* monitor string length *)
// 				IF LEN(CTRL.PATH) + LEN(CTRL.ELEMENT) + 1 > 250 THEN
// 					path_overflow := TRUE;
// 					CTRL.PATH := 'OVERFLOW';
// 				ELSE
// 					CTRL.PATH := CONCAT(CTRL.PATH,'/');
// 					CTRL.PATH  := CONCAT(CTRL.PATH,CTRL.ELEMENT);
// 				END_IF;
// 			END_IF;
//
// 			IF BIT_OF_DWORD(WORD_TO_DWORD(COMMAND),CTRL.TYP) THEN
//         				(*####################  DEBUG-MESSAGE  ###################################*)
//         				(*IF _debug_enable THEN
//           				LOG_CL.NEW_MSG := 'EL: #T:~1 #C:~2 #E:~3 #P:~6 #L:~7';
//           				LOG_CL.PRINTF[1] := INT_TO_STRING(CTRL.TYP);
//           				LOG_CL.PRINTF[2] := UINT_TO_STRING(CTRL.COUNT);
//           				LOG_CL.PRINTF[3] := CTRL.ELEMENT;
//           				LOG_CL.PRINTF[6] := CTRL.PATH;
//           				LOG_CL.PRINTF[7] := UINT_TO_STRING(CTRL.LEVEL);
//           				LOG_MSG();
//         				END_IF;*)
//         				(*########################################################################*)
// 				RETURN;
// 			END_IF;
// 		END_IF;
//
// 	200: (* ---------- TEXT SECTION ------------------ *)
// 		CTRL.VALUE := '';
// 		IF empty_tag = FALSE THEN
// 			s1 := index;
// 			(* search '<' end tag*)
// 			WHILE (index <= stop) AND (BUF[index] <> BYTE#60) DO
// 				index := index + 1;
// 			END_WHILE;
//
// 			E1 := index - 1;
// 			CTRL.BLOCK1_START := INT_TO_UINT(s1);
// 			CTRL.BLOCK1_STOP  := INT_TO_UINT(e1);
// 			CTRL.VALUE := BUFFER_TO_STRING(PT:=REF(BUF),SIZE:=INT_TO_UINT(stop + 1),START:=CTRL.BLOCK1_START,STOP:=CTRL.BLOCK1_STOP);
// 		END_IF;
//
// 		empty_tag := FALSE;
// 		mode := 300; (* -> NEXT-JOB: END ELEMENT *)
// 		CTRL.COUNT := CTRL.COUNT + UINT#1;
// 		CTRL.TYP := 3;
//
// 		IF BIT_OF_DWORD(WORD_TO_DWORD(command),CTRL.TYP) THEN
//       			(*####################  DEBUG-MESSAGE  ###################################*)
//       			(*IF _debug_enable THEN
//         				LOG_CL.NEW_MSG := 'TE: #T:~1 #C:~2 #E:~3 #V:~4 #P:~6 #L:~7';
//         				LOG_CL.PRINTF[1] := INT_TO_STRING(CTRL.TYP);
//         				LOG_CL.PRINTF[2] := UINT_TO_STRING(CTRL.COUNT);
//         				LOG_CL.PRINTF[3] := CTRL.ELEMENT;
//         				LOG_CL.PRINTF[4] := CTRL.VALUE;
//         				LOG_CL.PRINTF[6] := CTRL.PATH;
//         				LOG_CL.PRINTF[7] := UINT_TO_STRING(CTRL.LEVEL);
//         				LOG_MSG();
//       			END_IF;*)
//       			(*########################################################################*)
// 			RETURN;
// 		END_IF;
//
// 	300: (* ---------- END ELEMENT SECTION ------------------ *)
// 		WHILE (index <= stop) DO
// 			c := BUF[index];
// 			IF c = BYTE#62 THEN (* '>' TagEnd *)
// 				index := index + 1;
// 				s1 := FINDB(str1:=CTRL.PATH,str2:='/');
// 				IF path_overflow = FALSE THEN
// 					IF s1 > 1 THEN
// 						CTRL.ELEMENT := RIGHT(CTRL.PATH,LEN(CTRL.PATH) - s1);
// 						CTRL.PATH := LEFT(CTRL.PATH,s1 - 1);
// 					ELSE
// 						CTRL.ELEMENT := RIGHT(CTRL.PATH,LEN(CTRL.PATH) - 1);
// 						CTRL.PATH :='';
// 					END_IF;
// 				END_IF;
//
// 				CTRL.LEVEL := CTRL.LEVEL - UINT#1;
// 				CTRL.COUNT := CTRL.COUNT + UINT#1;
// 				CTRL.TYP := 2;
// 				mode := 100;
//
// 				IF BIT_OF_DWORD(WORD_TO_DWORD(COMMAND),CTRL.TYP) THEN
//          	 				(*####################  DEBUG-MESSAGE  ###################################*)
//           				(*IF _debug_enable THEN
//             					LOG_CL.NEW_MSG := 'CE: #T:~1 #C:~2 #E:~3 #P:~6 #L:~7';
//             					LOG_CL.PRINTF[1] := INT_TO_STRING(CTRL.TYP);
//             					LOG_CL.PRINTF[2] := UINT_TO_STRING(CTRL.COUNT);
//             					LOG_CL.PRINTF[3] := CTRL.ELEMENT;
//             					LOG_CL.PRINTF[6] := CTRL.PATH;
//             					LOG_CL.PRINTF[7] := UINT_TO_STRING(CTRL.LEVEL);
//             					LOG_MSG();
//           				END_IF;*)
//           				(*########################################################################*)
// 					RETURN;
// 				ELSE
// 					EXIT;
// 				END_IF;
// 			END_IF;
// 			index := index + 1;
// 		END_WHILE;
//
// 	400: (* ---------- ATTRIBUTE SECTION ------------------ *)
// 		(* search first normal charakter *)
// 		WHILE (index <= stop AND BUF[index] <= BYTE#32) DO
// 			index := index + 1;
// 		END_WHILE;
//
// 		(* begin Attribe name *)
// 		e1 := 0;
// 		s1 := index;
// 		(* search end of Attrib Name '=' *)
// 		WHILE (index <= stop) DO
// 			IF BUF[index] = BYTE#61 THEN (* '=' Equals *)
// 				e1 := index - 1;
// 				EXIT;
// 			END_IF;
// 			index := index + 1;
// 		END_WHILE;
//
// 		IF e1 > 0 THEN
// 			(* Attribute Name *)
// 			CTRL.BLOCK1_START := INT_TO_UINT(s1);
// 			CTRL.BLOCK1_STOP  := INT_TO_UINT(e1);
// 			CTRL.ATTRIBUTE := BUFFER_TO_STRING(PT:=REF(BUF),SIZE:=INT_TO_UINT(STOP + 1),START:=CTRL.BLOCK1_START,STOP:=CTRL.BLOCK1_STOP);
// 			(* search end of Attrib Value '=' *)
// 			index := index + 2;
// 			e1 := 0;
// 			s1 := INDEX;
// 			WHILE (index <= stop AND e1 = 0) DO
// 				c := BUF[index];
// 				IF c = BYTE#34 OR c = BYTE#39 THEN (* " OR ' Equals *)
// 					e1 := index - 1;
// 				END_IF;
// 				index := index + 1;
// 			END_WHILE;
//
// 			IF e1 > 0 THEN
// 				(* Value *)
// 				CTRL.BLOCK2_START := INT_TO_UINT(s1);
// 				CTRL.BLOCK2_STOP  := INT_TO_UINT(e1);
//
// 				(* for empty "" start is greater than stop and so it becomes an empty string *)
// 				CTRL.VALUE := BUFFER_TO_STRING(PT:=REF(BUF),SIZE:=INT_TO_UINT(stop + 1),START:=CTRL.BLOCK2_START,STOP:=CTRL.BLOCK2_STOP);
// 				(* search next non white space charakter *)
// 				WHILE (index <= stop AND BUF[index] <= BYTE#32) DO
// 					index := index + 1;
// 				END_WHILE;
//
// 					c := BUF[index];
// 					(* TagEnd '>' *)
// 					IF c = BYTE#62 THEN
// 						index := index + 1;
// 						index2 := index;
//
// 					(* search next non white space charakter *)
// 					WHILE (index <= stop AND BUF[index] <= BYTE#32) DO
// 						index := index + 1;
// 					END_WHILE;
//
// 					IF BUF[index] = BYTE#60 THEN (* TagBegin '<' *)
// 						mode := 100; (* -> NEXT-JOB: ELEMENT-SECTION *)
// 					ELSE
// 						index := index2;
// 						mode := 200; (* -> NEXT-JOB: TEXT-SECTION *)
// 					END_IF;
//
// 				ELSIF c = BYTE#47 OR c = BYTE#63 THEN (* TagTerm '/' OR '?' end Processing Instruction *)
// 					mode := 300; (* -> NEXT-JOB: END ELEMENT *)
// 				ELSE
// 					mode := 400; (* -> NEXT-JOB: ATTRIBUTE-SECTION *)
// 				END_IF;
//
// 				CTRL.COUNT := CTRL.COUNT + UINT#1;
// 				CTRL.TYP := 4;
// 				IF BIT_OF_DWORD(WORD_TO_DWORD(command),CTRL.TYP) THEN
//           				(*####################  DEBUG-MESSAGE  ###################################*)
//           				(*IF _debug_enable THEN
//             					LOG_CL.NEW_MSG := 'AT: #T:~1 #C:~2 #E:~3 #A:~4 #V:~5 #P:~6 #L:~7';
//             					LOG_CL.PRINTF[1] := INT_TO_STRING(CTRL.TYP);
//             					LOG_CL.PRINTF[2] := UINT_TO_STRING(CTRL.COUNT);
//             					LOG_CL.PRINTF[3] := CTRL.ELEMENT;
//             					LOG_CL.PRINTF[4] := CTRL.ATTRIBUTE;
//             					LOG_CL.PRINTF[5] := CTRL.VALUE;
//             					LOG_CL.PRINTF[6] := CTRL.PATH;
//             					LOG_CL.PRINTF[7] := UINT_TO_STRING(CTRL.LEVEL);
//             					LOG_MSG();
//           				END_IF;*)
//           				(*########################################################################*)
// 					RETURN;
// 				END_IF;
// 			END_IF;
// 		END_IF;
//
// 	500: (* ---------- SPECIAL DATA SECTION (Document Type Declarations) ---------- *)
//
// 		CTRL.TYP := 0;
// 		s1 := 0;
// 		index2 := 11;
//
// 		WHILE (s1 = 0) DO
// 			index2 := index2 + 1;
// 			CTRL.TYP := index2;
//
// 			CASE index2 OF
// 			12: (* CDATA *)
// 				s_code := '[CDATA[';
// 				e_code := ']]>';
// 			13: (* COMMENT *)
// 				s_code := '--';
// 				e_code := '-->';
// 			14: (* ANY DTD *)
// 				e_code := '';
// 				s1 := index;
// 				EXIT;
// 			END_CASE;
//
// 			e1 := LEN(s_code);
// 			IF BUFFER_SEARCH(PT:=REF(BUF),SIZE:=INT_TO_UINT(index + e1),STR:=S_CODE,POS:=index,IGN:=FALSE) = INDEX THEN
// 				s1 := index + e1;
// 			END_IF;
// 		END_WHILE;
//
// 		CTRL.BLOCK1_START := INT_TO_UINT(s1);
// 		IF LEN(e_code) > 0 THEN
// 			(* search end marker *)
// 			e1 := BUFFER_SEARCH(PT:=REF(BUF),SIZE:=INT_TO_UINT(stop + 1),STR:=e_code,POS:=index,IGN:=FALSE);
// 			CTRL.BLOCK1_STOP := INT_TO_UINT(e1 - 1);
// 			index := e1 + LEN(e_code); (* next element *)
// 		ELSE
// 			(* search '>' end tag*)
// 			index2 := 1; (* <> pair counter *)
// 			WHILE (index <= stop AND index2 > 0) DO
// 				c := BUF[index];
// 				IF c = BYTE#60 THEN (* '<' TagBegin *)
// 					index2 := index2 + 1;
// 				ELSIF c = BYTE#62 THEN (* '>' TagEnd   *)
// 					index2 := index2 - 1;
// 				ELSIF c = BYTE#34 OR c = BYTE#39 THEN (* " Double Quote OR ' Single Quote *)
// 					index := index + 1;
// 					WHILE (index <= stop) DO
// 						c := BUF[index];
// 						IF c = BYTE#34 OR c = BYTE#39 THEN (* " Double Quote OR ' Single Quote *)
// 							EXIT;
// 						END_IF;
// 						index := index + 1;
// 					END_WHILE;
// 				END_IF;
// 				index := index + 1;
// 			END_WHILE;
// 			CTRL.BLOCK1_STOP := INT_TO_UINT(index - 2);
// 		END_IF;
//
// 		CTRL.VALUE := BUFFER_TO_STRING(PT:=REF(BUF),SIZE:=INT_TO_UINT(stop + 1),START:=CTRL.BLOCK1_START,STOP:=CTRL.BLOCK1_STOP);
// 		CTRL.COUNT := CTRL.COUNT + UINT#1;
// 		mode := 100; (* -> NEXT-JOB: ELEMENT *)
//
// 		IF BIT_OF_DWORD(WORD_TO_DWORD(command),CTRL.TYP) THEN
//       			(*####################  DEBUG-MESSAGE  ###################################*)
//       			(*IF _debug_enable THEN
//         				LOG_CL.NEW_MSG := 'DTD: #T:~1 #C:~2 #S:~3 #E:~4 #V:~5 #P:~6 #L:~7';
//         				LOG_CL.PRINTF[1] := INT_TO_STRING(CTRL.TYP);
//         				LOG_CL.PRINTF[2] := UINT_TO_STRING(CTRL.COUNT);
//         				LOG_CL.PRINTF[3] := UINT_TO_STRING(CTRL.BLOCK1_START);
//         				LOG_CL.PRINTF[4] := UINT_TO_STRING(CTRL.BLOCK1_STOP);
//         				LOG_CL.PRINTF[5] := CTRL.VALUE;
//         				LOG_CL.PRINTF[6] := CTRL.PATH;
//         				LOG_CL.PRINTF[7] := UINT_TO_STRING(CTRL.LEVEL);
//         				LOG_MSG();
//       			END_IF;*)
//       			(*########################################################################*)
// 			RETURN;
// 		END_IF;
//
// 	END_CASE;
// END_WHILE;
// END_FUNCTION_BLOCK

// Commented out for beedance: it uses FLOAT_TO_REAL, which is commented out.
// FUNCTION_BLOCK YAHOO_WEATHER
// VAR_IN_OUT
// 	IP_C : IP_C; (* IP_Control management structure *)
// 	S_BUF : NETWORK_BUFFER;
// 	R_BUF : NETWORK_BUFFER;
// 	YW : YAHOO_WEATHER_DATA;
// END_VAR
// VAR_INPUT
// 	ACTIVATE : BOOL;
// 	UNITS : BOOL;
// 	LOCATION : STRING(20);
// END_VAR
// VAR_OUTPUT
// 	BUSY : BOOL;
// 	DONE : BOOL;
// 	ERROR_C : DWORD;
// 	ERROR_T : BYTE;
// END_VAR
// VAR
// 	CTRL : XML_CONTROL;
// 	XML_READER : XML_READER;
// 	URL_DATA : url;
// 	DNS_CLIENT : DNS_CLIENT;
// 	HTTP_GET : HTTP_GET;
// 	activate_last : BOOL;
// 	value_int : INT;
// 	value_real : REAL;
// 	v_real : REAL;
// 	state : INT;
// 	cycle : INT;
// 	day_idx :	INT;
// 	idx : INT;
// 	cnt :	INT;
//
// 	(*
// 	_debug_state_last : INT := -1;
// 	_debug_enable : BOOL := TRUE;
// 	LOG_MSG : LOG_MSG;
// 	*)
// END_VAR
//
// CASE state OF
//
// 00:	IF ACTIVATE AND NOT activate_last THEN
// 		state := 40;
// 		DONE := FALSE;
// 		BUSY := TRUE;
// 		ERROR_C := DWORD#0;
// 		ERROR_T := BYTE#0;
// 		cycle := 0;
//   		URL_DATA.DOMAIN := 'query.yahooapis.com'; (* domain name for DNS_CLIENT *)
// 	END_IF;
//
// 40:	IF DNS_CLIENT.DONE THEN
// 		state := 50;
// 	ELSIF (DNS_CLIENT.ERROR > DWORD#00) THEN
// 		(* error handling *)
// 		ERROR_C := DNS_CLIENT.ERROR;
// 	ERROR_T := BYTE#01;
// 		state   := 100;
// 	END_IF;
//
// 50:   	(* Teil 1: http://query.yahooapis.com/v1/public/yql?q=select%20units,wind,atmosphere,astronomy,location%20from%20weather.forecast%20where%20woeid=551801%20AND%20u=%27c%27
//              part 2: http://query.yahooapis.com/v1/public/yql?q=select%20item%20from%20weather.forecast%20where%20woeid=551801%20AND%20u=%27c%27 *)
//
// 	IF cycle = 0 THEN
//   		URL_DATA.QUERY := 'q=select%20units,wind,atmosphere,astronomy,location%20from%20weather.forecast%20where%20woeid='; (* part 1 - infos *)
//   	ELSE
//   		URL_DATA.QUERY := 'q=select%20item%20from%20weather.forecast%20where%20woeid='; (* part 2 - daily data *)
//   	END_IF;
//
//   	URL_DATA.QUERY := CONCAT(URL_DATA.QUERY,LOCATION); (* location *)
//
//   	IF UNITS THEN
//     		URL_DATA.QUERY := CONCAT(URL_DATA.QUERY,'%20and%20u=%27f%27'); (* fahrenheit *)
//   	ELSE
//     		URL_DATA.QUERY := CONCAT(URL_DATA.QUERY,'%20and%20u=%27c%27'); (* celsius *)
//   	END_IF;
//
//   	URL_DATA.PATH := '/v1/public/yql';
//
//   	state := 60;
//
// 60:	IF HTTP_GET.DONE THEN
// 		state := 80;
// 		CTRL.START_POS := HTTP_GET.BODY_START;
// 		CTRL.STOP_POS := HTTP_GET.BODY_STOP;
// 		CTRL.COMMAND := WORD#2#10000000_00011000; (* ONLY TEXT AND ATTRIBUTE *)
// 		CTRL.WATCHDOG  := T#1ms;
//
// 	ELSIF (HTTP_GET.ERROR > DWORD#00) THEN
// 		(* error handling *)
// 		ERROR_C := HTTP_GET.ERROR;
// 		ERROR_T := BYTE#02;
// 		state := 100;
// 	END_IF;
//
// 80: XML_READER(CTRL:=CTRL,BUF:=R_BUF.BUFFER); (* read XML data serially *)
// 	IF CTRL.TYP < 98 THEN (* evaluate only if not a watchdog pass *)
// 		value_int := 0;
// 		value_real := 0.0;
// 		(* perform automatic conversion to real and int *)
// 		IF LEN(CTRL.VALUE) <= 20 THEN
// 			v_real:=FLOAT_TO_REAL(FLT:=CTRL.VALUE);
// 			IF CHK_REAL(v_real) = 0 THEN (* !!! checks for a valid REAL value, otherwise TwinCAT 2.x can crash !!!!  *)
// 				value_real := v_real;
// 				value_int := REAL_TO_INT(value_real);
// 			END_IF;
// 		END_IF;
//
// 		(*####################  DEBUG-MESSAGE  ###################################*)
// 		(*IF _debug_enable THEN
// 			LOG_CL.NEW_MSG := 'XML: ~2 # ~3 # ~4 # ~5';
// 			LOG_CL.PRINTF[2] := UINT_TO_STRING(CTRL.LEVEL);
// 			LOG_CL.PRINTF[3] := UINT_TO_STRING(CTRL.COUNT);
// 			LOG_CL.PRINTF[4] := CTRL.ELEMENT;
// 			LOG_CL.PRINTF[5] := CTRL.VALUE;
// 			LOG_MSG();
// 		END_IF;*)
// 		(*########################################################################*)
//
// 		IF cycle = 0 THEN
// 	      		(* ------------ part 1 --------------*)
// 	      		CASE UINT_TO_INT(CTRL.COUNT) OF
// 	        		014: YW.location_city := CTRL.VALUE;
// 	        		015: YW.location_country := CTRL.VALUE;
// 	        		016: YW.location_region := CTRL.VALUE;
// 	        		020: YW.wind_chill := value_int;
// 	        		021: YW.wind_direction := value_int;
// 	        		022: YW.wind_speed := value_real;
// 	        		026: YW.atmosphere_humidity := value_int;
// 	        		027: YW.atmosphere_pressure := value_real;
// 	        		028: YW.atmosphere_rising := value_int;
// 	        		029: YW.atmosphere_visibility := value_real;
// 	        		033: YW.astronomy_sunrise := CTRL.VALUE;
// 	        		034: YW.astronomy_sunset := CTRL.VALUE;
// 	        		038: YW.unit_distance := CTRL.VALUE;
// 	        		039: YW.unit_pressure := CTRL.VALUE;
// 	        		040: YW.unit_speed := CTRL.VALUE;
// 	        		041: YW.unit_temperature := CTRL.VALUE;
// 	      		END_CASE;
// 	    	ELSE
// 	      		(* ------------ part 2 --------------*)
// 	      		CASE UINT_TO_INT(CTRL.COUNT) OF
// 	        		018: YW.GEO_LATITUDE := value_real;
// 	        		022: YW.GEO_LONGITUDE := value_real;
//
// 			032: YW.CUR_CONDITIONS_CODE := value_int;
// 			         YW.CUR_CONDITIONS_ICON := value_int;
// 	        		034: YW.CUR_CONDITIONS_TEMP := value_int;
// 	        		035: YW.CUR_CONDITIONS_TEXT := CTRL.VALUE;
//
// 			039: YW.FORECAST_TODAY_CODE := value_int;
// 			         YW.FORECAST_TODAY_ICON := value_int;
// 			040: YW.FORECAST_TODAY_DATE_LONG := CTRL.VALUE;
// 	        		042: YW.FORECAST_TODAY_HIGH_TEMP := value_int;
// 	        		043: YW.FORECAST_TODAY_LOW_TEMP := value_int;
// 	        		044: YW.FORECAST_TODAY_TEXT := CTRL.VALUE;
//
// 			048..125: (* forcast day 1-10 *)
// 				cnt := UINT_TO_INT(CTRL.COUNT) - 48;
// 				day_idx := cnt / 9 + 1;
// 				idx := cnt MOD 9;
// 	      	  		CASE idx OF
// 					0:	YW.FORECAST_DAY[day_idx].CODE := value_int;
// 						YW.FORECAST_DAY[day_idx].ICON := value_int;
// 					1:	YW.FORECAST_DAY[day_idx].DATE_LONG := CTRL.VALUE;
// 					3:	YW.FORECAST_DAY[day_idx].HIGH_TEMP := value_int;
// 					4:	YW.FORECAST_DAY[day_idx].LOW_TEMP := value_int;
// 					5:	YW.FORECAST_DAY[day_idx].TEXT := CTRL.VALUE;
// 	      	  		END_CASE;
// 	      		END_CASE;
// 	    	END_IF;
// 	ELSIF CTRL.TYP = 99 THEN (* EXIT - last element read *)
// 		state := 100;
// 	END_IF;
//
// 100:	(* UNLOCK HTTP DATA *)
// 	IF (NOT HTTP_GET.DONE) THEN
// 		IF cycle = 0 AND ERROR_T = BYTE#0 THEN
// 			(* run part 2 *)
//     			state := 50;
// 			cycle := cycle + 1;
// 		ELSE
// 	    		state := 0;
// 	    		BUSY  := FALSE;
// 	    		DONE := ERROR_T = BYTE#0;
// 		END_IF;
// 	END_IF;
//
// END_CASE;
//
// (* ---------------- DNS --------------- *)
// DNS_CLIENT(	IP_C:=IP_C,
// 			S_BUF:=S_BUF,
// 			R_BUF:=R_BUF,
// 			DOMAIN:=URL_DATA.DOMAIN,
// 			IP4_DNS:=DWORD#00,
// 			ACTIVATE:=state=40 (* DNS Start *)
// 			);
// (* parameters not used, or not used directly *)
// (*	DWORD :=DNS_CLIENT.IP4;
// 	BOOL  :=DNS_CLIENT.DONE;
// 	BYTE  :=DNS_CLIENT.ERROR; *)
// (* -------------------------------------*)
//
// (* ------------- HTTP_GET --------------- *)
// HTTP_GET(	IP_C:=IP_C,
// 			S_BUF:=S_BUF,
// 			R_BUF:=R_BUF,
// 			IP4:=DNS_CLIENT.IP4,
// 			GET:=state=60,
// 			MODE:=BYTE#2, (* HTTP 1.1 with persistent connection *)
// 			UNLOCK_BUF:=state=100,
// 			URL_DATA:=URL_DATA
// 			);
//
// (* parameters not used, or not used directly *)
// (*	STRING := HTTP_GET.HTTP_STATUS;
// 	UINT :=HTTP_GET.HEADER_START;
// 	UINT :=HTTP_GET.HEADER_STOP;
// 	UINT :=HTTP_GET.BODY_START;
// 	UINT :=HTTP_GET.BODY_STOP;
// 	BOOL :=HTTP_GET.DONE;
// 	BYTE :=HTTP_GET.ERROR;
// *)
// (* -------------------------------------*)
//
// activate_last := ACTIVATE;
//
// (*####################  DEBUG-MESSAGE  ###################################*)
// (*IF _debug_enable THEN
// 	IF state <> _debug_state_last THEN
// 		LOG_CL.NEW_MSG := 'yw-step: /last ~1 /New ~2';
// 		LOG_CL.PRINTF[1] := INT_TO_STRING(_debug_state_last);
// 		LOG_CL.PRINTF[2] := INT_TO_STRING(state);
// 		LOG_MSG();
// 		_debug_state_last := state;
// 	END_IF;
// END_IF;*)
// (*########################################################################*)
// END_FUNCTION_BLOCK

FUNCTION_BLOCK YAHOO_WEATHER_DESC_GE
VAR_IN_OUT
	YW : YAHOO_WEATHER_DATA;
END_VAR
VAR_INPUT
	ACTIVATE : BOOL;
END_VAR
VAR
	act_last : BOOL;
	x : INT;
	y : INT;
	str : STRING(40);
END_VAR

IF ACTIVATE AND act_last = FALSE THEN
	FOR y := 1 TO 12 DO
		CASE y OF
		01:	x := YW.CUR_CONDITIONS_CODE;

		02:	YW.CUR_CONDITIONS_TEXT := str;
			x := YW.FORECAST_TODAY_CODE;
		03:	YW.FORECAST_TODAY_TEXT := str;
			x := YW.FORECAST_DAY[1].CODE;
		04:	YW.FORECAST_DAY[1].TEXT := str;
			x := YW.FORECAST_DAY[2].CODE;
		05:	YW.FORECAST_DAY[2].TEXT := str;
			x := YW.FORECAST_DAY[3].CODE;
		06:	YW.FORECAST_DAY[3].TEXT := str;
			x := YW.FORECAST_DAY[4].CODE;
		07:	YW.FORECAST_DAY[4].TEXT := str;
			x := YW.FORECAST_DAY[5].CODE;
		08:	YW.FORECAST_DAY[5].TEXT := str;
			x := YW.FORECAST_DAY[6].CODE;
		09:	YW.FORECAST_DAY[6].TEXT := str;
			x := YW.FORECAST_DAY[7].CODE;
		10:	YW.FORECAST_DAY[7].TEXT := str;
			x := YW.FORECAST_DAY[8].CODE;
		11:	YW.FORECAST_DAY[8].TEXT := str;
			x := YW.FORECAST_DAY[9].CODE;
		12:	YW.FORECAST_DAY[9].TEXT := str;
		END_CASE;

		CASE x OF
		00:	str := 'Wirbelsturm';
		01:	str := 'Tropensturm';
		02:	str := 'Wirbelsturm';
		03:	str := 'starkes Gewitter ';
		04:	str := 'Gewitter';
		05:	str := 'Schneeregen';
		06:	str := 'Schneeregen';
		07:	str := 'Schneeregen';
		08:	str := 'gefrierender Nieselregen';
		09:	str := 'Nieselregen';
		10:	str := 'gefrierender Regen';
		11:	str := 'Regenfälle';
		12:	str := 'Regenfälle';
		13:	str := 'Schneegestöber';
		14:	str := 'leichte Schneefälle';
		15:	str := 'Schneetreiben';
		16:	str := 'Schnee';
		17:	str := 'Hagel';
		18:	str := 'Schneeregen';
		19:	str := 'Staub';
		20:	str := 'nebelig';
		21:	str := 'Dunst';
		22:	str := 'rauchig';
		23:	str := 'stürmisch';
		24:	str := 'windig';
		25:	str := 'kalt';
		26:	str := 'bewölkt';
		27:	str := 'meist bewölkt';
		28:	str := 'meist bewölkt';
		29:	str := 'teilweise bewölkt';
		30:	str := 'teilweise bewölkt';
		31:	str := 'klar';
		32:	str := 'sonnig';
		33:	str := 'heiter';
		34:	str := 'heiter';
		35:	str := 'Regen und Hagel';
		36:	str := 'heiß';
		37:	str := 'örtliche Gewitter';
		38:	str := 'vereinzelte Gewitter';
		39:	str := 'vereinzelte Gewitter';
		40:	str := 'vereinzelte Regenfälle';
		41:	str := 'schwere Schneefälle';
		42:	str := 'vereinzelte Schneefälle';
		43:	str := 'schwere Schneefälle';
		44:	str := 'teilweise bewölkt';
		45:	str := 'gewittrige Regenfälle';
		46:	str := 'Schneefälle';
		47:	str := 'örtliche gewittrige Regenfälle';
		ELSE
			str := 'nicht verfügbar';
		END_CASE;
	END_FOR;
END_IF;
act_last := ACTIVATE;
END_FUNCTION_BLOCK

FUNCTION_BLOCK YAHOO_WEATHER_ICON_OSCAT
VAR_IN_OUT
	YW : YAHOO_WEATHER_DATA;
END_VAR
VAR_INPUT
	ACTIVATE : BOOL;
END_VAR
VAR
	dat : ARRAY[0..48] OF INT := 4,2,2,4,17,1,3,1,2,2,2,2,2,3,3,3,3,5,3,6,7,14,8,9,9,10,9,11,12,11,12,13,14,15,16,4,14,4,17,2,2,3,3,3,12,2,3,4,0;
	act_last : BOOL;
	x : INT;
	idx : INT;
END_VAR

IF ACTIVATE AND act_last = FALSE THEN
	x := MIN(YW.CUR_CONDITIONS_CODE,48);
	YW.CUR_CONDITIONS_ICON := dat[x];
	x := MIN(YW.FORECAST_TODAY_CODE,48);
	YW.FORECAST_TODAY_ICON := dat[x];
	FOR idx := 1 TO 9 DO
		x := MIN(YW.FORECAST_DAY[idx].CODE,48);
		YW.FORECAST_DAY[idx].ICON := dat[x];
	END_FOR;
END_IF;
act_last := ACTIVATE;
END_FUNCTION_BLOCK

TYPE DLOG_CRON_DATA :
STRUCT
	CE : ARRAY [0..5] OF DLOG_CRON_ELEMENT;
END_STRUCT
END_TYPE

TYPE DLOG_CRON_ELEMENT :
STRUCT
	ELEMENTS : ARRAY [0..59] OF BOOL;
	VALUE : INT;
	VALUE_MIN : INT;
	VALUE_MAX : INT;
	ALL_SELECTED : BOOL;
END_STRUCT
END_TYPE

TYPE DLOG_DATA :
STRUCT
	STORE_TYPE : BYTE;
	ADD_COM : INT;
	ADD_DATA_REQ : BOOL;
	CLOCK_TRIG : BOOL;
	ID_MAX : USINT;
	DTI : DT;
	UCB : UNI_CIRCULAR_BUFFER_DATA;
	LOAD_TIME_MAX : TIME;
	NEW_FILE : STRING;
	NEW_FILE_SIZE : UDINT;
	NEW_FILE_RTRIG : BOOL;
END_STRUCT
END_TYPE

TYPE
	DLOG_REAL_ARRAY_DATA : ARRAY [1..64] OF DLOG_REAL_ARRAY_ELEMENT;
END_TYPE

TYPE DLOG_REAL_ARRAY_ELEMENT :
STRUCT
	VALUE : REAL;
	DELTA : REAL;
	COLUMN : STRING(10);
	_DELTA_LAST : 	REAL;
	_VALUE_LAST : 	REAL;
END_STRUCT
END_TYPE

TYPE DLOG_RETAIN :
STRUCT
	FN_REM : STRING;
	COLOR : BOOL;
	HEAD: BOOL;
	TRIG_CNT : UDINT;
	TRIG_CNT_TOTAL : UDINT;
END_STRUCT
END_TYPE

TYPE DLOG_SAVE :
STRUCT
	FN_REM : STRING;
	COLOR : BOOL;
	HEAD: BOOL;
	TRIG_CNT : UDINT;
	TRIG_CNT_TOTAL : UDINT;
END_STRUCT
END_TYPE

TYPE FILE_PATH_DATA :
STRUCT
	DRIVE : STRING(3);
	DIRECTORY : STRING(STRING_LENGTH);
	FILENAME : STRING;
END_STRUCT
END_TYPE

TYPE FILE_SERVER_DATA :
STRUCT
	FILE_OPEN : BOOL;
	FILENAME : STRING;
	MODE : BYTE;
	OFFSET : UDINT;
	FILE_SIZE : UDINT;
	ERROR : BYTE;
	RUNTIME : FILE_SERVER_RUNTIME_DATA;
END_STRUCT
END_TYPE

TYPE FILE_SERVER_RUNTIME_DATA :
STRUCT
	TIME_FILE_OPEN_CUR : UDINT;
	TIME_FILE_OPEN_MAX : UDINT;
	TIME_FILE_OPEN_MIN : UDINT;
	TIME_FILE_CLOSE_CUR : UDINT;
	TIME_FILE_CLOSE_MAX : UDINT;
	TIME_FILE_CLOSE_MIN : UDINT;
	TIME_FILE_READ_CUR: UDINT;
	TIME_FILE_READ_MAX : UDINT;
	TIME_FILE_READ_MIN : UDINT;
	TIME_FILE_WRITE_CUR : UDINT;
	TIME_FILE_WRITE_MAX : UDINT;
	TIME_FILE_WRITE_MIN : UDINT;
	TIME_FILE_SEEK_CUR : UDINT;
	TIME_FILE_SEEK_MAX : UDINT;
	TIME_FILE_SEEK_MIN : UDINT;
	TIME_FILE_TELL_CUR : UDINT;
	TIME_FILE_TELL_MAX : UDINT;
	TIME_FILE_TELL_MIN : UDINT;
	TIME_FILE_DELETE_CUR : UDINT;
	TIME_FILE_DELETE_MAX : UDINT;
	TIME_FILE_DELETE_MIN : UDINT;
END_STRUCT
END_TYPE

TYPE IP2GEO_DATA :
STRUCT
	STATE : BOOL;
	IP4 : DWORD;
	COUNTRY_CODE : STRING(2);
	COUNTRY_NAME : STRING(20);
	REGION_CODE : STRING(2);
	REGION_NAME : STRING(20);
	CITY : STRING(20);
	GEO_LATITUDE : REAL;
	GEO_LONGITUDE : REAL;
	TIME_ZONE_NAME : STRING(20);
	GMT_OFFSET : INT;
	IS_DST : BOOL;
END_STRUCT
END_TYPE

TYPE IP_C :
STRUCT
	C_MODE : BYTE;						(*W Mode: TCP/UDP ACTIVE/PASSIVE                               *)
	C_PORT : WORD;						(*W port number                                               *)
	C_IP : DWORD;						(*W IP address packed wwxxyyzz = www.xxx.yyy.zzz            *)
	C_STATE : BYTE;						(*R connection status ON/OFF + edge ON/OFF                 *)
	C_ENABLE : BOOL;					(*W enable for connect                                     *)
	R_OBSERVE : BOOL;					(*W monitor receive                                      *)
	TIME_RESET : BOOL;					(*W reset all timers                                   *)
	ERROR : DWORD;					(*R vvwwxxyy (vv = CON_ERROR, ww = SEN_ERROR, xx = REC_ERROR *)
	FIFO : IP_FIFO_DATA;					(*I IP FIFO structure                                         *)
	MAILBOX : ARRAY [1..16] OF BYTE;	(*I mailbox: data area for data exchange between blocks         *)
END_STRUCT
END_TYPE

TYPE IP_FIFO_DATA :
STRUCT
	X : ARRAY [1..128] OF BYTE; 	(* IP_ID FIFO memory          *)
	Y : ARRAY [1..128] OF BYTE; 	(* IP_ID counter                 *)
	ID : BYTE;					(* highest assigned id         *)
	MAX_ID : BYTE;				(* maximum registrations per ID   *)
	INIT : BOOL;					(* initialization done *)
	EMPTY : BOOL;				(* FIFO empty                    *)
	FULL : BOOL;					(* FIFO full                    *)
	TOP : INT;					(* maximum number in FIFO      *)
	NW : INT;					(* write pointer                *)
	NR : INT;						(* read pointer                   *)
END_STRUCT
END_TYPE

TYPE LOG_CONTROL :
STRUCT
	NEW_MSG : STRING(LOG_SIZE); (* new message for the data buffer *)
	NEW_MSG_OPTION : DWORD;
	LEVEL : BYTE;
	SIZE : INT := LOG_MAX; (* number of strings in LOG_DATA *)
	RESET : BOOL; (* clear message buffer *)
	PRINTF : PRINTF_DATA; (* Array PRINTF Parameter *)
	MSG : ARRAY [0..LOG_MAX] OF STRING(LOG_SIZE); (* Array Message *)
	MSG_OPTION : ARRAY [0..LOG_MAX] OF DWORD; (* Array Options *)
	UPDATE_COUNT : UINT; (* update counter *)
	IDX : INT; (* current message index *)
	RING_MODE : BOOL; (* buffer overflow detected *)
END_STRUCT
END_TYPE

TYPE MYSQL_COM :
STRUCT
	S_BUF : NETWORK_BUFFER;
	R_BUF : NETWORK_BUFFER;
	SQL_CON : BOOL;
	SQL_URL : STRING(STRING_LENGTH);
	SQL_PACKET_NO : BYTE;
	TIMEOUT : TIME;
	DNS_IP4 : DWORD;
	SQL_RCV_STATE : BYTE;
	ERROR_C : DWORD;
	ERROR_T : BYTE;
END_STRUCT
END_TYPE

TYPE MYSQL_INFO :
STRUCT
	SERVER_PROTOCOL_VERSION : BYTE;
	SERVER_CAPABILITIES : WORD;
	SERVER_STATUS : WORD;
	SERVER_LANGUAGE : BYTE;
	SQL_CONNECTED : BOOL;
	SQL_ERROR : STRING(STRING_LENGTH);
	DATA_INSERT_AKTIV : BOOL;
	DATA_INSERT_OK_CNT : UDINT;
	DATA_INSERT_NOK_CNT : UDINT;
END_STRUCT
END_TYPE

TYPE NET_VAR_DATA :
STRUCT
	CYCLE : UDINT;
	STATE : BYTE;
	INDEX : INT;
	ID_MAX : USINT;
	ERROR_ID : BYTE;
	BUF_SIZE : UINT;
	S_BUF : NETWORK_BUFFER;
	R_BUF : NETWORK_BUFFER;
END_STRUCT
END_TYPE

TYPE NETWORK_BUFFER :
STRUCT
	SIZE : UINT;
	BUFFER : NW_BUF_LONG;
END_STRUCT
END_TYPE

TYPE NETWORK_BUFFER_SHORT :
STRUCT
	SIZE : UINT;
	BUFFER : NW_BUF_SHORT;
END_STRUCT
END_TYPE

TYPE
	NW_BUF_LONG  : ARRAY[0..NETWORK_BUFFER_LONG_SIZE] OF BYTE;
END_TYPE

TYPE
	NW_BUF_SHORT : ARRAY[0..NETWORK_BUFFER_SHORT_SIZE] OF BYTE;
END_TYPE

TYPE PRINTF_DATA : ARRAY [1..11]  OF STRING(LOG_SIZE);
END_TYPE

TYPE
	UNI_CIRCULAR_BUF : ARRAY [0..8191] OF BYTE;
END_TYPE

TYPE UNI_CIRCULAR_BUFFER_DATA :
STRUCT
	D_MODE : INT;
	D_SIZE : INT;
	D_HEAD : WORD;
	D_STRING : STRING(STRING_LENGTH);
	D_REAL : REAL;
	D_DWORD : DWORD;
	BUF_SIZE : UINT;
	BUF_COUNT : UINT;
	BUF_USED : USINT;
	BUF_USED_MAX : USINT;
	BUF_DATA_CNT : UDINT;
	BUF_DATA_LOST : UDINT;
	BUF : UNI_CIRCULAR_BUF;
	_GetStart : UINT;
	_GetEnd : UINT;
	_Last : UINT;
	_First : UINT;
END_STRUCT
END_TYPE

TYPE URL :
STRUCT
	PROTOCOL : STRING(10);
	USER : STRING(32);
	PASSWORD : STRING(32);
	DOMAIN : STRING(80);
	PORT : WORD;
	PATH : STRING(80);
	QUERY : STRING(STRING_LENGTH);
	ANCHOR : STRING(40);
	HEADER : STRING(160);
END_STRUCT
END_TYPE

TYPE us_LOG_VIEWPORT :
STRUCT
	LINE_ARRAY : ARRAY [1..40] OF INT;
	COUNT : INT; (* number of visible messages *)
	UPDATE_COUNT : UINT; (* update counter *)
	MOVE_TO_X : INT; (* control of the message display *)
	UPDATE : BOOL; (* data was changed -> redraw *)
END_STRUCT
END_TYPE

TYPE us_TN_INPUT_CONTROL :
STRUCT
	bo_Enable: BOOL; (* enable/disable processing *)
	bo_Update_all: BOOL; (* redraw all elements *)
	bo_Reset_Fokus: BOOL; (* set focus on 1st element *)
	in_Focus_at: INT; (* control element with active focus *)
	in_Count: INT; (* number of used control elements *)
	in_ToolTip_X: INT; (* Tooltip Text X-Offset *)
	in_ToolTip_Y: INT; (* Tooltip Text Y-Offset *)
	by_ToolTip_Attr: BYTE; (* Tooltip Text Attribute *)
	in_ToolTip_Size: INT; (* tooltip text length *)
	usa_TN_INPUT_CONTROL_DATA: ARRAY [1..20] OF us_TN_INPUT_CONTROL_DATA;
END_STRUCT
END_TYPE

TYPE us_TN_INPUT_CONTROL_DATA :
STRUCT
 	by_Input_Exten_Code: BYTE;
	by_Input_ASCII_Code: BYTE;
	bo_Input_ASCII_IsNum: BOOL;
	in_Title_X_Offset: INT; (* Title Text X-Offset *)
	in_Title_Y_Offset: INT; (* Title Text Y-Offset *)
	by_Title_Attr: BYTE; (* Title Text Attribute *)
	st_Title_String: STRING; (* Title Text String *)
	in_Cursor_X: INT; (* current cursor X position *)
	in_Cursor_Y: INT; (* current cursor Y position *)
	in_Type: INT; (* type of the element *)
	in_X: INT; (* Element X-Position *)
	in_Y: INT; (* Element Y-Position *)
	in_Cursor_Pos: INT; (* current cursor position *)
	by_Attr_mF: BYTE; (* text attributes with focus *)
	by_Attr_oF: BYTE; (* text attributes without focus *)
	in_selected: INT; (* text item was selected *)
	st_Input_Mask: STRING; (* text input mask *)
	st_Input_Data: STRING(STRING_LENGTH); (* text current input data *)
	st_Input_String: STRING; (* text copy after return key *)
	st_Input_ToolTip: STRING; (* text tooltip (input information) *)
	in_Input_Option: INT; (* text output options *)
	bo_Input_Entered: BOOL; (* RETURN key was pressed *)
	bo_Input_Hidden: BOOL; (* text hidden input with '*' *)
	bo_Input_Only_Num: BOOL; (* text allow numeric input only *)
	bo_Focus: BOOL; (* element has the focus *)
	bo_Update_Input: BOOL; (* redraw element because of user input *)
	bo_Update_All: BOOL; (* redraw element completely *)

END_STRUCT
END_TYPE

TYPE us_TN_MENU :
STRUCT
	st_Menu_Text: STRING(STRING_LENGTH); (* X menu texts *)
	in_Menu_E_Count: INT; (* menu element count *)
	in_Y: INT; (* menu line number  Y position *)
	in_X: INT; (* menu column number X position *)
	by_Attr_mF: BYTE; (* text attributes with focus *)
	by_Attr_oF: BYTE; (* text attributes without focus *)
	in_X_SM_new: INT; (* new submenu X position *)
	in_Y_SM_new: INT; (* new submenu Y position *)
	in_X_SM_old: INT; (* old submenu X position *)
	in_Y_SM_old: INT; (* old submenu Y position *)
	in_Cur_Menu_Item: INT; (* current main menu *)
	in_Cur_Sub_Item: INT; (* current submenu *)
	in_State: INT; (*   Menu status   *)
	in_Menu_Selected: INT; (* X menu item selected with enter *)
	bo_Create: BOOL; (* X create menu *)
	bo_Destroy: BOOL; (* X remove menu *)
	bo_Update: BOOL; (* X update menu *)
END_STRUCT
END_TYPE

TYPE us_TN_MENU_POPUP :
STRUCT
	st_Menu_Text: STRING(STRING_LENGTH); (* X menu texts *)
	in_Menu_E_Count: INT; (* menu element count *)
	in_X: INT; (* X menu X position *)
	in_Y: INT; (* X menu Y position *)
	in_Cols: INT; (* menu column count *)
	in_Rows: INT; (* menu line count *)
	in_Cur_Item: INT; (* X current submenu *)
	by_Attr_mF: BYTE; (* X text attributes with focus	*)
	by_Attr_oF: BYTE; (* X text attributes without focus *)
	by_Input_Exten_Code: BYTE; (* X key code: special keys *)
	bo_Create: BOOL; (* X create popup menu *)
	bo_Destroy: BOOL; (* X remove popup menu *)
	bo_Update: BOOL; (* X update popup menu *)
	bo_Activ: BOOL; (*   popup menu is active *)
END_STRUCT
END_TYPE
